// TIA Portal project "JAN0837_proof_of_concept" (V20)

(* hardware
DEVICE "R2D2"  S7-1200 Station
   slot 0: "Rack_0"  S7-1200 Rack  Rack  V1.0
   slot 1: "R2D2_Sharp7"  CPU 1212C DC/DC/DC  6ES7 212-1AE40-0XB0  V4.6
DEVICE "R2D2_1"  S7-1200 Station
   slot 0: "Rack_0"  S7-1200 Rack  Rack  V1.0
   slot 1: "R2D2_OPCUA"  CPU 1212C DC/DC/DC  6ES7 212-1AE40-0XB0  V4.6
DEVICE "R2D2_2"  S7-1200 Station
   slot 0: "Rack_0"  S7-1200 Rack  Rack  V1.0
   slot 1: "R2D2_MQTT"  CPU 1212C DC/DC/DC  6ES7 212-1AE40-0XB0  V4.6
DEVICE "R2D2_3"  S7-1200 Station
   slot 0: "Rack_0"  S7-1200 Rack  Rack  V1.0
   slot 1: "R2D2_MODBUS"  CPU 1212C DC/DC/DC  6ES7 212-1AE40-0XB0  V4.6
DEVICE "R2D2_4"  S7-1200 Station
   slot 0: "Rack_0"  S7-1200 Rack  Rack  V1.0
   slot 1: "R2D2_RESTAPI"  CPU 1212C DC/DC/DC  6ES7 212-1AE40-0XB0  V4.6
*)

// ===== PLC "R2D2_Sharp7"  CPU 1212C DC/DC/DC =====

VAR_GLOBAL   // PLC tag table "Default tag table"
   "Clock_Byte" AT %MB0 : Byte;
   "Clock_10Hz" AT %M0.0 : Bool;
   "Clock_5Hz" AT %M0.1 : Bool;
   "Clock_2.5Hz" AT %M0.2 : Bool;
   "Clock_2Hz" AT %M0.3 : Bool;
   "Clock_1.25Hz" AT %M0.4 : Bool;
   "Clock_1Hz" AT %M0.5 : Bool;
   "Clock_0.625Hz" AT %M0.6 : Bool;
   "Clock_0.5Hz" AT %M0.7 : Bool;
   "System_Byte" AT %MB1 : Byte;
   "FirstScan" AT %M1.0 : Bool;
   "DiagStatusUpdate" AT %M1.1 : Bool;
   "AlwaysTRUE" AT %M1.2 : Bool;
   "AlwaysFALSE" AT %M1.3 : Bool;
END_VAR

VAR_GLOBAL   // PLC tag table "Regulator"
   "Regulator_PV" AT %MD100 : Real;
   "Regulator_SetPoint" AT %MD104 : Real;
END_VAR

VAR_GLOBAL   // PLC tag table "CarLight"
   "CarLight_Tag1" AT %M50.0 : Bool;
END_VAR

VAR_GLOBAL   // PLC tag table "Crossroad"
   "Crossroad_Tag_1" AT %M300.0 : Bool;
   "Crossroad_Tag_2" AT %M300.1 : Bool;
   "Crossroad_Tag_3" AT %MW302 : Word;
   "Crossroad_MEM 0" AT %M304.0 : Bool;
   "Crossroad_MEM 1" AT %M304.1 : Bool;
   "Crossroad_MEM 2" AT %M304.2 : Bool;
   "Crossroad_MEM 3" AT %M304.3 : Bool;
   "Crossroad_MEM 4" AT %M304.4 : Bool;
   "Crossroad_MEM 5" AT %M304.5 : Bool;
   "Crossroad_Clock" AT %MW328 : Int;
   "Crossroad_DayModeState" AT %MB305 : USInt;
   "Crossroad_ActualLengthState" AT %MD316 : Time;
   "Crossorad_HoursDayStart" AT %MW320 : Int;
   "Crossroad_HoursDayEnd" AT %MW322 : Int;
   "Crossroad_DayStarts" AT %MW324 : Int;
   "Crossroad_DayEnds" AT %MW326 : Int;
   "Crossroad_S1" AT %MB306 : USInt;
   "Crossroad_S2" AT %MB307 : USInt;
   "Crossroad_S3" AT %MB308 : USInt;
   "Crossroad_S4" AT %MB309 : USInt;
   "Crossroad_S5" AT %MB310 : USInt;
   "Crossroad_S6" AT %MB311 : USInt;
   "Crossroad_S7" AT %MB312 : USInt;
   "Crossroad_S8" AT %MB313 : USInt;
   "Crossroad_S9" AT %MB314 : USInt;
   "Crossroad_Walk_EN" AT %M330.0 : Bool;
END_VAR

VAR_GLOBAL   // PLC tag table "Crosswalk"
   "Crosswalk_CTU_current_value" AT %MW200 : Int;
   "Crosswalk_CTU_reset" AT %M202.0 : Bool;
   "Crosswalk_DayMode" AT %M202.1 : Bool;
   "Crosswalk_NightMode" AT %M202.2 : Bool;
   "Crosswalk_OffMode" AT %M202.3 : Bool;
   "Crosswalk_DaySeq" AT %MW204 : Int;
   "Crosswalk_NightSeq" AT %MW206 : Int;
END_VAR

TYPE "Crossroad_Input"
   STRUCT
      btnStart : Bool := FALSE;
      btnPause : Bool := FALSE;
      btnStop : Bool := FALSE;
      btnWestCrosswalk1 : Bool := FALSE;
      btnWestCrosswalk2 : Bool := FALSE;
      btnSouthCrosswalk1 : Bool := FALSE;
      btnSouthCrosswalk2 : Bool := FALSE;
      spare1 : DWord := 0;
      spare2 : DWord := 0;
      spare3 : DWord := 0;
      spare4 : DWord := 0;
   END_STRUCT;
END_TYPE

TYPE "Crossroad_Output"
   STRUCT
      crossroadType : Bool := FALSE;
      trafficLightNorth_green : Bool := FALSE;
      trafficLightNorth_yellow : Bool := FALSE;
      trafficLightNorth_red : Bool := FALSE;
      trafficLightSouth_green : Bool := FALSE;
      trafficLightSouth_yellow : Bool := FALSE;
      trafficLightSouth_red : Bool := FALSE;
      trafficLightWest_green : Bool := FALSE;
      trafficLightWest_yellow : Bool := FALSE;
      trafficLightWest_red : Bool := FALSE;
      trafficLightEast_green : Bool := FALSE;
      trafficLightEast_yellow : Bool := FALSE;
      trafficLightEast_red : Bool := FALSE;
      pedestrianSouth1_green : Bool := FALSE;
      pedestrianSouth1_red : Bool := FALSE;
      pedestrianSouth2_green : Bool := FALSE;
      pedestrianSouth2_red : Bool := FALSE;
      pedestrianWest1_green : Bool := FALSE;
      pedestrianWest1_red : Bool := FALSE;
      pedestrianWest2_green : Bool := FALSE;
      pedestrianWest2_red : Bool := FALSE;
      spare1 : DWord := 0;
      spare2 : DWord := 0;
      spare3 : DWord := 0;
      spare4 : DWord := 0;
   END_STRUCT;
END_TYPE

TYPE "Crosswalk_Input"
   STRUCT
      btnStart : Bool := FALSE;
      btnPause : Bool := FALSE;
      btnStop : Bool := FALSE;
      btnCrosswalk1 : Bool := FALSE;
      btnCrosswalk2 : Bool := FALSE;
      spare1 : DWord := 0;
      spare2 : DWord := 0;
      spare3 : DWord := 0;
      spare4 : DWord := 0;
   END_STRUCT;
END_TYPE

TYPE "Crosswalk_Output"
   STRUCT
      crosswalkType : Bool := FALSE;
      trafficLightGreen1 : Bool := FALSE;
      trafficLightsYellow1 : Bool := FALSE;
      trafficLightsRed1 : Bool := FALSE;
      trafficLightGreen2 : Bool := FALSE;
      trafficLightsYellow2 : Bool := FALSE;
      trafficLightsRed2 : Bool := FALSE;
      pedestrianLightGreen1 : Bool := FALSE;
      pedestrianLightRed1 : Bool := FALSE;
      pedestrianLightGreen2 : Bool := FALSE;
      pedestrianLightRed2 : Bool := FALSE;
      spare1 : DWord := 0;
      spare2 : DWord := 0;
      spare3 : DWord := 0;
      spare4 : DWord := 0;
   END_STRUCT;
END_TYPE

TYPE "Regulator_Input"
   STRUCT
      btnReset : Bool := FALSE;
      switchstate : Bool := FALSE;
      order : Int := 1;
      R1 : Real := 0.0;
      R2 : Real := 0.0;
      C1 : Real := 0.0;
      C2 : Real := 0.0;
      Uc1 : Real := 0.0;
      Uc2 : Real := 0.0;
      Td : Real := 0.0;
      Ts : Real := 0.0;
      spare1 : DWord := 0;
      spare2 : DWord := 0;
      spare3 : DWord := 0;
      spare4 : DWord := 0;
   END_STRUCT;
END_TYPE

TYPE "Regulator_Output"
   STRUCT
      Uin : Real := 0.0;
      spare1 : DWord := 0;
      spare2 : DWord := 0;
      spare3 : DWord := 0;
      spare4 : DWord := 0;
   END_STRUCT;
END_TYPE

TYPE "CarLight_Input"
   STRUCT
      btnReset : Bool := FALSE;
      error : Bool := FALSE;
      sensorLight : Bool := FALSE;
      sensorConnectorConnected : Bool := FALSE;
      result : Bool := FALSE;
      spare1 : DWord := 0;
      spare2 : DWord := 0;
      spare3 : DWord := 0;
      spare4 : DWord := 0;
   END_STRUCT;
END_TYPE

TYPE "CarLight_Output"
   STRUCT
      lowBeamLight : Bool := FALSE;
      highBeamLight : Bool := FALSE;
      turnLight : Bool := FALSE;
      spare1 : DWord := 0;
      spare2 : DWord := 0;
      spare3 : DWord := 0;
      spare4 : DWord := 0;
   END_STRUCT;
END_TYPE

DATA_BLOCK "DB_ProcessData"   // DB1
{ S7_Optimized_Access := 'TRUE' }
VERSION : 0.1
   VAR
      crossroad_input : "Crossroad_Input";
      crossroad_output : "Crossroad_Output";
      crosswalk_input : "Crosswalk_Input";
      crosswalk_output : "Crosswalk_Output";
      regulator_input : "Regulator_Input";
      regulator_output : "Regulator_Output";
      carlight_input : "CarLight_Input";
      carlight_output : "CarLight_Output";
   END_VAR
BEGIN
END_DATA_BLOCK

// folder: CarLight

DATA_BLOCK "CarLight_SCL_DB"   // DB12
{ S7_Optimized_Access := 'TRUE' }
VERSION : 0.1
// stored: InstanceOfName CarLight_SCL
"CarLight_SCL"
BEGIN
END_DATA_BLOCK

// folder: System blocks/Program resources

DATA_BLOCK "IEC_Counter_0_DB"   // DB2
{ S7_Optimized_Access := 'TRUE' }
AUTHOR : Simatic
FAMILY : IEC
NAME : CNTR
VERSION : 1.0
// stored: InstanceOfName IEC_COUNTER
"IEC_COUNTER"
BEGIN
END_DATA_BLOCK

DATA_BLOCK "IEC_Timer_0_DB"   // DB3
{ S7_Optimized_Access := 'TRUE' }
AUTHOR : Simatic
FAMILY : IEC
NAME : IEC_TMR
VERSION : 1.0
// stored: InstanceOfName IEC_TIMER
"IEC_TIMER"
BEGIN
END_DATA_BLOCK

DATA_BLOCK "IEC_Timer_CrosswalkGreen_DB_1"   // DB4
{ S7_Optimized_Access := 'TRUE' }
AUTHOR : Simatic
FAMILY : IEC
NAME : IEC_TMR
VERSION : 1.0
// stored: InstanceOfName IEC_TIMER
"IEC_TIMER"
BEGIN
END_DATA_BLOCK

DATA_BLOCK "IEC_Timer_CrosswalkYellow1_DB_1"   // DB5
{ S7_Optimized_Access := 'TRUE' }
AUTHOR : Simatic
FAMILY : IEC
NAME : IEC_TMR
VERSION : 1.0
// stored: InstanceOfName IEC_TIMER
"IEC_TIMER"
BEGIN
END_DATA_BLOCK

DATA_BLOCK "IEC_Timer_CrosswalkRed_DB_1"   // DB6
{ S7_Optimized_Access := 'TRUE' }
AUTHOR : Simatic
FAMILY : IEC
NAME : IEC_TMR
VERSION : 1.0
// stored: InstanceOfName IEC_TIMER
"IEC_TIMER"
BEGIN
END_DATA_BLOCK

DATA_BLOCK "IEC_Timer_CrosswalkYellow2_DB_1"   // DB7
{ S7_Optimized_Access := 'TRUE' }
AUTHOR : Simatic
FAMILY : IEC
NAME : IEC_TMR
VERSION : 1.0
// stored: InstanceOfName IEC_TIMER
"IEC_TIMER"
BEGIN
END_DATA_BLOCK

DATA_BLOCK "IEC_Timer_CrosswalkOn_DB_1"   // DB8
{ S7_Optimized_Access := 'TRUE' }
AUTHOR : Simatic
FAMILY : IEC
NAME : IEC_TMR
VERSION : 1.0
// stored: InstanceOfName IEC_TIMER
"IEC_TIMER"
BEGIN
END_DATA_BLOCK

DATA_BLOCK "IEC_Timer_CrosswalkOff_DB_1"   // DB9
{ S7_Optimized_Access := 'TRUE' }
AUTHOR : Simatic
FAMILY : IEC
NAME : IEC_TMR
VERSION : 1.0
// stored: InstanceOfName IEC_TIMER
"IEC_TIMER"
BEGIN
END_DATA_BLOCK

DATA_BLOCK "IEC_Timer_CrossroadCycle_DB_1"   // DB10
{ S7_Optimized_Access := 'TRUE' }
AUTHOR : Simatic
FAMILY : IEC
NAME : IEC_TMR
VERSION : 1.0
// stored: InstanceOfName IEC_TIMER
"IEC_TIMER"
BEGIN
END_DATA_BLOCK

// folder: (top level)

ORGANIZATION_BLOCK "Main"   // OB1, LAD, ProgramCycle
TITLE = "Main Program Sweep (Cycle)"
{ S7_Optimized_Access := 'TRUE' }
VERSION : 0.1
   VAR_INPUT
      Initial_Call : Bool;   // Initial call of this OB
      Remanence : Bool;   // =True, if remanent data are available
   END_VAR
BEGIN

REGION Network 1: CarLight
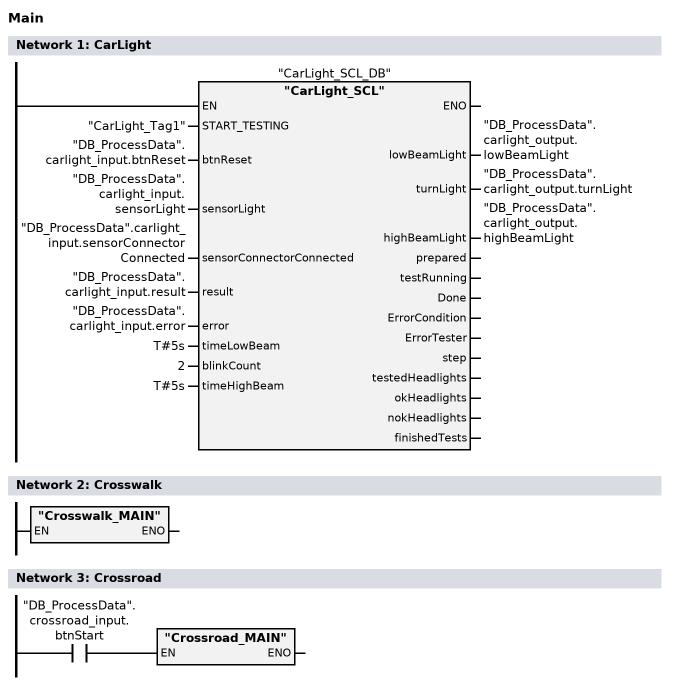
   RUNG wire#powerrail
      "CarLight_SCL_DB"(START_TESTING := "CarLight_Tag1", btnReset := "DB_ProcessData".carlight_input.btnReset, sensorLight := "DB_ProcessData".carlight_input.sensorLight, sensorConnectorConnected := "DB_ProcessData".carlight_input.sensorConnectorConnected, result := "DB_ProcessData".carlight_input.result, error := "DB_ProcessData".carlight_input.error, timeLowBeam := T#5s, blinkCount := 2, timeHighBeam := T#5s, lowBeamLight => "DB_ProcessData".carlight_output.lowBeamLight, turnLight => "DB_ProcessData".carlight_output.turnLight, highBeamLight => "DB_ProcessData".carlight_output.highBeamLight, prepared =>, testRunning =>, Done =>, ErrorCondition =>, ErrorTester =>, "step" =>, testedHeadlights =>, okHeadlights =>, nokHeadlights =>, finishedTests =>)
   END_RUNG
   // the same network as SCL:
   "CarLight_SCL_DB"(START_TESTING := "CarLight_Tag1",   // "CarLight_SCL"
                     btnReset := "DB_ProcessData".carlight_input.btnReset,
                     sensorLight := "DB_ProcessData".carlight_input.sensorLight,
                     sensorConnectorConnected := "DB_ProcessData".carlight_input.sensorConnectorConnected,
                     result := "DB_ProcessData".carlight_input.result,
                     error := "DB_ProcessData".carlight_input.error,
                     timeLowBeam := T#5s,
                     blinkCount := 2,
                     timeHighBeam := T#5s,
                     lowBeamLight => "DB_ProcessData".carlight_output.lowBeamLight,
                     turnLight => "DB_ProcessData".carlight_output.turnLight,
                     highBeamLight => "DB_ProcessData".carlight_output.highBeamLight);
END_REGION

REGION Network 2: Crosswalk
   RUNG wire#powerrail
      "Crosswalk_MAIN"()
   END_RUNG
   // the same network as SCL:
   "Crosswalk_MAIN"();
END_REGION

REGION Network 3: Crossroad
   RUNG wire#powerrail
      Contact( "DB_ProcessData".crossroad_input.btnStart )
      "Crossroad_MAIN"()
   END_RUNG
   // the same network as SCL:
   IF "DB_ProcessData".crossroad_input.btnStart THEN "Crossroad_MAIN"(); END_IF;
END_REGION
END_ORGANIZATION_BLOCK

ORGANIZATION_BLOCK "CyclicInterrupt"   // OB30, LAD, CyclicInterrupt
{ S7_Optimized_Access := 'TRUE' }
VERSION : 0.1
   VAR_INPUT
      Initial_Call : Bool;   // Initial call of this OB
      Event_Count : Int;   // Events discarded
   END_VAR
BEGIN

REGION Network 1: Regulator
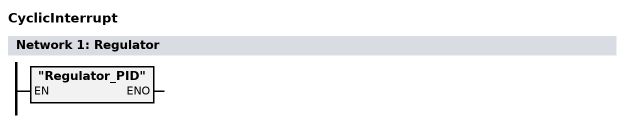
   RUNG wire#powerrail
      "Regulator_PID"()
   END_RUNG
   // the same network as SCL:
   "Regulator_PID"();
END_REGION
END_ORGANIZATION_BLOCK

ORGANIZATION_BLOCK "Startup"   // OB100, LAD, Startup
TITLE = "Complete Restart"
{ S7_Optimized_Access := 'TRUE' }
VERSION : 0.1
   VAR_INPUT
      LostRetentive : Bool;   // True if retentive data are lost
      LostRTC : Bool;   // True if date and time are lost
   END_VAR
BEGIN

REGION Network 1 (SCL)
   // Communication 


   // Crossroad
   "Crossorad_HoursDayStart" := 0;
   "Crossroad_HoursDayEnd" := 2400;
   "Crossroad_DayStarts" := 500;
   "Crossroad_DayEnds" := 2200;
   "Crossroad_S1" := 1;
   "Crossroad_S2" := 2;
   "Crossroad_S3" := 3;
   "Crossroad_S4" := 4;
   "Crossroad_S5" := 5;
   "Crossroad_S6" := 6;
   "Crossroad_S7" := 7;
   "Crossroad_S8" := 8;
   "Crossroad_S9" := 9;


   // Crosswalk


   // Regulaotr


   // CarLight
END_REGION
END_ORGANIZATION_BLOCK

// folder: CarLight

FUNCTION_BLOCK "CarLight_SCL"   // FB1, SCL
{ S7_Optimized_Access := 'TRUE' }
VERSION : 0.1
   VAR_INPUT
      START_TESTING : Bool;
      btnReset : Bool;
      sensorLight : Bool;
      sensorConnectorConnected : Bool;
      result : Bool;
      error : Bool;
      timeLowBeam : Time;
      blinkCount : Int;
      timeHighBeam : Time;
   END_VAR
   VAR_OUTPUT
      lowBeamLight : Bool;
      turnLight : Bool;
      highBeamLight : Bool;
      prepared : Bool;
      testRunning : Bool;
      Done : Bool;
      ErrorCondition : Bool;
      ErrorTester : Bool;
      "step" : Int;
      testedHeadlights : DInt;
      okHeadlights : DInt;
      nokHeadlights : DInt;
      finishedTests : DInt;
   END_VAR
   VAR
      state : Int;
      ready : Bool;
      start_old : Bool;
      start_rise : Bool;
      conditionsErrorLatched : Bool;
      testerErrorLatched : Bool;
      blinkTarget : Int;
      blinkIndex : Int;
      resultStored : Bool;
      testerResponseSeenTrue : Bool;
      tonLowBeam : TON_TIME;
      tonBlinkOn : TON_TIME;
      tonBlinkOff : TON_TIME;
      tonHighBeam : TON_TIME;
      tonAll : TON_TIME;
      tonTesterResponse : TON_TIME;
   END_VAR
BEGIN
   // ---------------------------------------------------------------------
   // Helper signals
   // ---------------------------------------------------------------------
   #ready := #sensorLight AND #sensorConnectorConnected;

   IF #blinkCount < 1 THEN
       #blinkTarget := 1;
   ELSE
       #blinkTarget := #blinkCount;
   END_IF;

   #start_rise := #START_TESTING AND NOT #start_old;
   #start_old := #START_TESTING;


   // ---------------------------------------------------------------------
   // RESET process (counters are NOT cleared)
   // ---------------------------------------------------------------------
   IF #btnReset THEN
       #state := 0;
       #conditionsErrorLatched := FALSE;
       #testerErrorLatched := FALSE;   
       #blinkIndex := 0;
       #resultStored := FALSE;
       #testerResponseSeenTrue := FALSE;
   END_IF;


   // ---------------------------------------------------------------------
   // Loss of required conditions during test
   // ---------------------------------------------------------------------
   IF ((#state >= 20) AND (#state <= 55)) AND (NOT #ready) THEN
       #state := 0;
       #conditionsErrorLatched := TRUE;
       #blinkIndex := 0;
       #resultStored := FALSE;
       #testerResponseSeenTrue := FALSE;
   END_IF;


   // ---------------------------------------------------------------------
   // Tester error – immediate NOK termination
   // ---------------------------------------------------------------------
   IF ((#state >= 20) AND (#state <= 55)) AND #error THEN

       #testerErrorLatched := TRUE;

       IF NOT #resultStored THEN
           #testedHeadlights := #testedHeadlights + 1;
           #nokHeadlights := #nokHeadlights + 1;
           #resultStored := TRUE;
       END_IF;

       #blinkIndex := 0;
       #testerResponseSeenTrue := FALSE;

       #state := 70;

   END_IF;


   // ---------------------------------------------------------------------
   // State machine
   // ---------------------------------------------------------------------
   CASE #state OF


           // ==============================================================
           // 0 - IDLE
           // ==============================================================
       0:

           #lowBeamLight := FALSE;
           #turnLight := FALSE;
           #highBeamLight := FALSE;

           #tonLowBeam(IN := FALSE,
                     PT := #timeLowBeam);
           #tonBlinkOn(IN := FALSE,
                       PT := T#1s);
           #tonBlinkOff(IN := FALSE,
                        PT := T#1s);
           #tonHighBeam(IN := FALSE,
                     PT := #timeHighBeam);
           #tonAll(IN := FALSE,
                   PT := T#5s);
           #tonTesterResponse(IN := FALSE,
                              PT := T#1s);

           IF #start_rise THEN

               IF #ready AND (NOT #error) THEN

                   #conditionsErrorLatched := FALSE;
                   #testerErrorLatched := FALSE;
                   #blinkIndex := 0;
                   #resultStored := FALSE;
                   #testerResponseSeenTrue := FALSE;

                   #state := 20;

               ELSE

                   IF NOT #ready THEN
                       #conditionsErrorLatched := TRUE;
                   END_IF;

                   IF #error THEN
                       #testerErrorLatched := TRUE;
                   END_IF;

               END_IF;

           END_IF;


           // ==============================================================
           // 20 - LOW BEAM
           // ==============================================================
       20:

           #lowBeamLight := TRUE;
           #turnLight := FALSE;
           #highBeamLight := FALSE;

           #tonLowBeam(IN := TRUE,
                     PT := #timeLowBeam);
           #tonBlinkOn(IN := FALSE,
                       PT := T#1s);
           #tonBlinkOff(IN := FALSE,
                        PT := T#1s);
           #tonHighBeam(IN := FALSE,
                     PT := #timeHighBeam);
           #tonAll(IN := FALSE,
                   PT := T#5s);
           #tonTesterResponse(IN := FALSE,
                              PT := T#1s);

           IF #tonLowBeam.Q THEN
               #blinkIndex := 0;
               #state := 30;
           END_IF;


           // ==============================================================
           // 30 - TURN SIGNAL ON
           // ==============================================================
       30:

           #lowBeamLight := FALSE;
           #turnLight := TRUE;
           #highBeamLight := FALSE;

           #tonLowBeam(IN := FALSE,
                     PT := #timeLowBeam);
           #tonBlinkOn(IN := TRUE,
                       PT := T#1s);
           #tonBlinkOff(IN := FALSE,
                        PT := T#1s);
           #tonHighBeam(IN := FALSE,
                     PT := #timeHighBeam);
           #tonAll(IN := FALSE,
                   PT := T#5s);
           #tonTesterResponse(IN := FALSE,
                              PT := T#1s);

           IF #tonBlinkOn.Q THEN
               #state := 31;
           END_IF;


           // ==============================================================
           // 31 - TURN SIGNAL OFF
           // ==============================================================
       31:

           #lowBeamLight := FALSE;
           #turnLight := FALSE;
           #highBeamLight := FALSE;

           #tonLowBeam(IN := FALSE,
                     PT := #timeLowBeam);
           #tonBlinkOn(IN := FALSE,
                       PT := T#1s);
           #tonBlinkOff(IN := TRUE,
                        PT := T#1s);
           #tonHighBeam(IN := FALSE,
                     PT := #timeHighBeam);
           #tonAll(IN := FALSE,
                   PT := T#5s);
           #tonTesterResponse(IN := FALSE,
                              PT := T#1s);

           IF #tonBlinkOff.Q THEN

               #blinkIndex := #blinkIndex + 1;

               IF #blinkIndex < #blinkTarget THEN
                   #state := 30;
               ELSE
                   #state := 40;
               END_IF;

           END_IF;


           // ==============================================================
           // 40 - HIGH BEAM
           // ==============================================================
       40:

           #lowBeamLight := FALSE;
           #turnLight := FALSE;
           #highBeamLight := TRUE;

           #tonLowBeam(IN := FALSE,
                     PT := #timeLowBeam);
           #tonBlinkOn(IN := FALSE,
                       PT := T#1s);
           #tonBlinkOff(IN := FALSE,
                        PT := T#1s);
           #tonHighBeam(IN := TRUE,
                     PT := #timeHighBeam);
           #tonAll(IN := FALSE,
                   PT := T#5s);
           #tonTesterResponse(IN := FALSE,
                              PT := T#1s);

           IF #tonHighBeam.Q THEN
               #state := 50;
           END_IF;


           // ==============================================================
           // 50 - ALL LIGHTS (5 seconds)
           // ==============================================================
       50:

           #lowBeamLight := TRUE;
           #turnLight := TRUE;
           #highBeamLight := TRUE;

           #tonLowBeam(IN := FALSE,
                     PT := #timeLowBeam);
           #tonBlinkOn(IN := FALSE,
                       PT := T#1s);
           #tonBlinkOff(IN := FALSE,
                        PT := T#1s);
           #tonHighBeam(IN := FALSE,
                     PT := #timeHighBeam);
           #tonAll(IN := TRUE,
                   PT := T#5s);
           #tonTesterResponse(IN := FALSE,
                              PT := T#1s);

           IF #tonAll.Q THEN
               #testerResponseSeenTrue := FALSE;
               #state := 55;
           END_IF;


           // ==============================================================
           // 55 - WAIT 1 s FOR RESULT
           // ==============================================================
       55:

           #lowBeamLight := FALSE;
           #turnLight := FALSE;
           #highBeamLight := FALSE;

           #tonLowBeam(IN := FALSE,
                     PT := #timeLowBeam);
           #tonBlinkOn(IN := FALSE,
                       PT := T#1s);
           #tonBlinkOff(IN := FALSE,
                        PT := T#1s);
           #tonHighBeam(IN := FALSE,
                     PT := #timeHighBeam);
           #tonAll(IN := FALSE,
                   PT := T#5s);
           #tonTesterResponse(IN := TRUE,
                              PT := T#1s);

           IF #result THEN
               #testerResponseSeenTrue := TRUE;
           END_IF;

           IF #tonTesterResponse.Q THEN

               IF NOT #resultStored THEN

                   #testedHeadlights := #testedHeadlights + 1;

                   IF #testerResponseSeenTrue THEN
                       #okHeadlights := #okHeadlights + 1;
                   ELSE
                       #nokHeadlights := #nokHeadlights + 1;
                   END_IF;

                   #resultStored := TRUE;

               END_IF;

               #finishedTests := #finishedTests + 1;

               #state := 60;

           END_IF;


           // ==============================================================
           // 60 - FINISHED
           // ==============================================================
       60:

           #lowBeamLight := FALSE;
           #turnLight := FALSE;
           #highBeamLight := FALSE;

           IF #start_rise THEN

               IF #ready AND (NOT #error) THEN

                   #conditionsErrorLatched := FALSE;
                   #testerErrorLatched := FALSE;
                   #blinkIndex := 0;
                   #resultStored := FALSE;
                   #testerResponseSeenTrue := FALSE;

                   #state := 20;

               END_IF;

           END_IF;


           // ==============================================================
           // 70 - TESTER ERROR
           // ==============================================================
       70:

           #lowBeamLight := FALSE;
           #turnLight := FALSE;
           #highBeamLight := FALSE;

           IF #start_rise THEN

               IF #ready AND (NOT #error) THEN

                   #conditionsErrorLatched := FALSE;
                   #testerErrorLatched := FALSE;
                   #blinkIndex := 0;
                   #resultStored := FALSE;
                   #testerResponseSeenTrue := FALSE;

                   #state := 20;

               END_IF;

           END_IF;

       ELSE

           #state := 0;

   END_CASE;


   // ---------------------------------------------------------------------
   // State outputs
   // ---------------------------------------------------------------------
   #testRunning := (#state >= 20) AND (#state <= 55);

   #prepared := #ready AND (NOT #error) AND
   ((#state = 0) OR (#state = 60) OR (#state = 70));

   #Done := (#state = 60);

   #ErrorCondition := #conditionsErrorLatched;
   #ErrorTester := #testerErrorLatched;

   #step := #state;
END_FUNCTION_BLOCK

// folder: Crossroad

FUNCTION "Crossroad_MAIN" : Void   // FC4, LAD
{ S7_Optimized_Access := 'TRUE' }
VERSION : 0.1
   VAR_TEMP   // added for the SCL form of the ladder/FBD networks
      _w1 : Bool;
      _w2 : Bool;
      _w3 : Bool;
      _w4 : Bool;
   END_VAR
BEGIN

REGION Network 1: Time based decision process
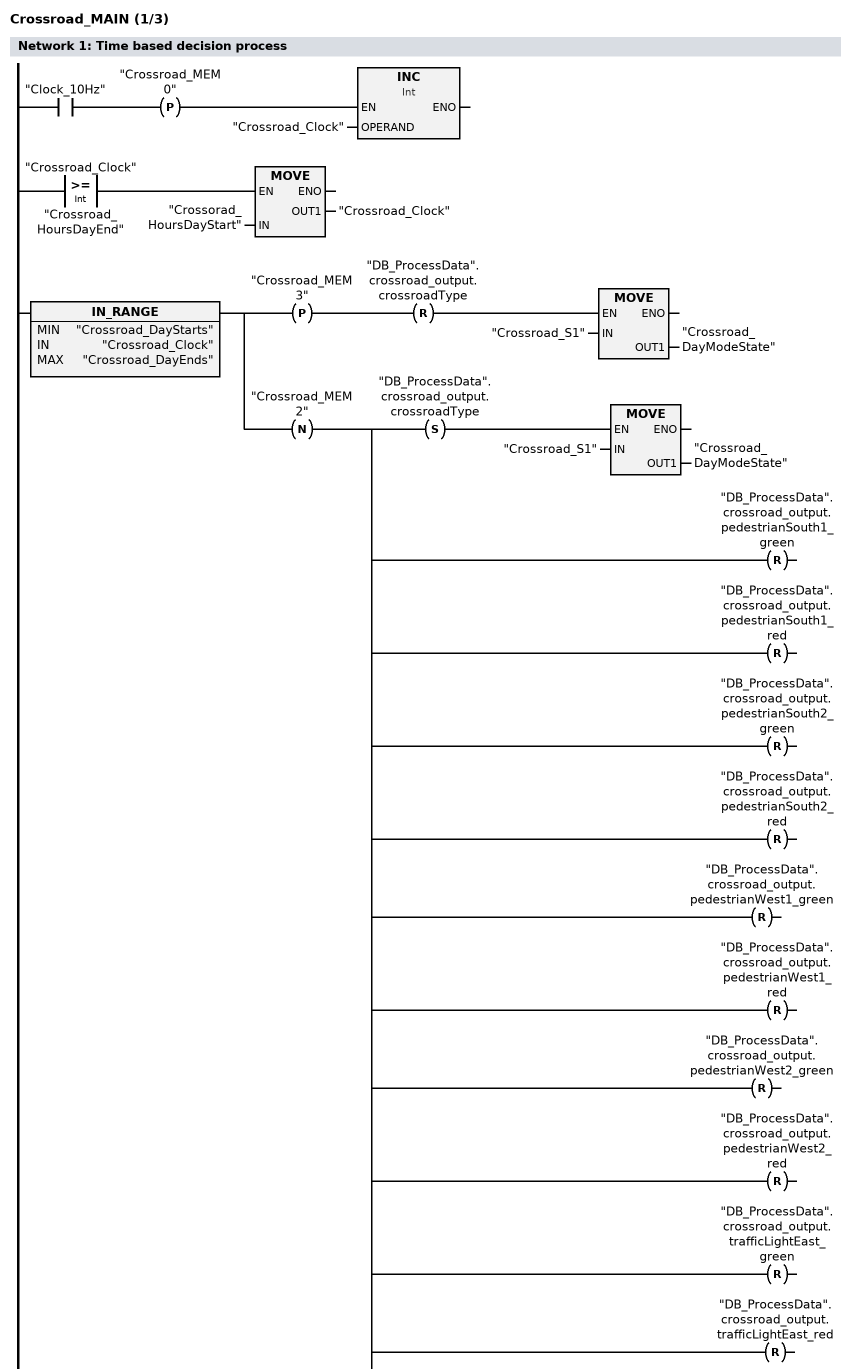
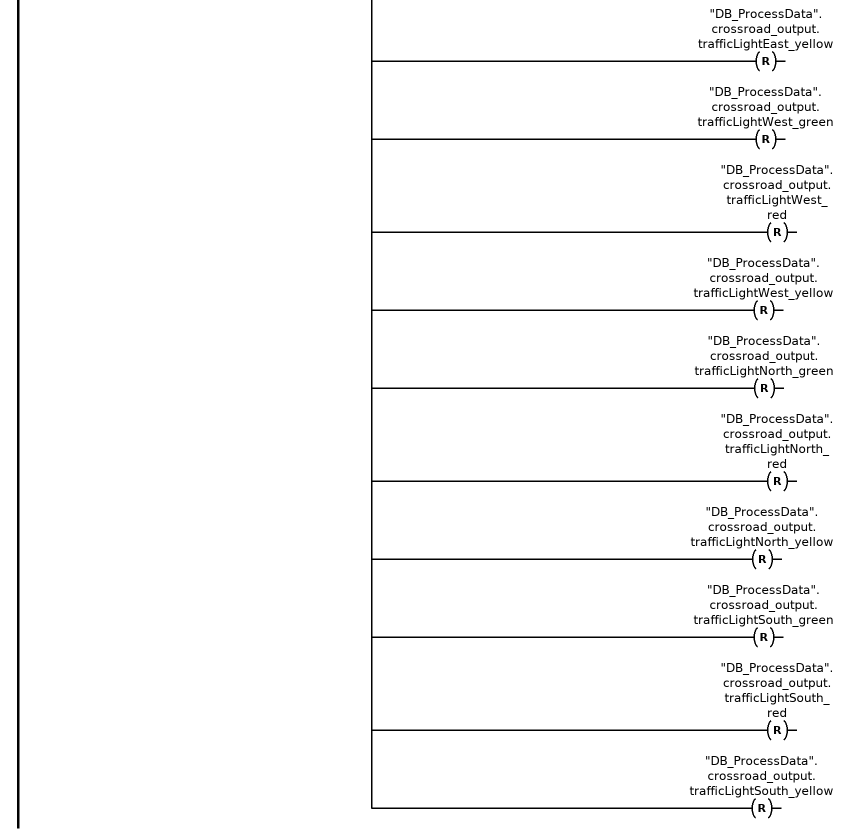
   RUNG wire#powerrail
      Contact( "Clock_10Hz" )
      P_Trig( "Crossroad_MEM 0" )
      { S7_Templates := "DestType := Int" } Inc( "Crossroad_Clock" )
   END_RUNG
   RUNG wire#powerrail
      { S7_Templates := "SrcType := Int" } GE_Contact(in1 := "Crossroad_Clock", in2 := "Crossroad_HoursDayEnd")
      Move(in := "Crossorad_HoursDayStart", out1 => "Crossroad_Clock")
   END_RUNG
   RUNG wire#powerrail
      { S7_Templates := "SrcType := Int" } InRange(min := "Crossroad_DayStarts", in := "Crossroad_Clock", max := "Crossroad_DayEnds")
      wire#w1
      P_Trig( "Crossroad_MEM 3" )
      R_Coil( "DB_ProcessData".crossroad_output.crossroadType )
      Move(in := "Crossroad_S1", out1 => "Crossroad_DayModeState")
   END_RUNG
   RUNG wire#w1
      N_Trig( "Crossroad_MEM 2" )
      wire#w2
      S_Coil( "DB_ProcessData".crossroad_output.crossroadType )
      Move(in := "Crossroad_S1", out1 => "Crossroad_DayModeState")
   END_RUNG
   RUNG wire#w2
      R_Coil( "DB_ProcessData".crossroad_output.pedestrianSouth1_green )
   END_RUNG
   RUNG wire#w2
      R_Coil( "DB_ProcessData".crossroad_output.pedestrianSouth1_red )
   END_RUNG
   RUNG wire#w2
      R_Coil( "DB_ProcessData".crossroad_output.pedestrianSouth2_green )
   END_RUNG
   RUNG wire#w2
      R_Coil( "DB_ProcessData".crossroad_output.pedestrianSouth2_red )
   END_RUNG
   RUNG wire#w2
      R_Coil( "DB_ProcessData".crossroad_output.pedestrianWest1_green )
   END_RUNG
   RUNG wire#w2
      R_Coil( "DB_ProcessData".crossroad_output.pedestrianWest1_red )
   END_RUNG
   RUNG wire#w2
      R_Coil( "DB_ProcessData".crossroad_output.pedestrianWest2_green )
   END_RUNG
   RUNG wire#w2
      R_Coil( "DB_ProcessData".crossroad_output.pedestrianWest2_red )
   END_RUNG
   RUNG wire#w2
      R_Coil( "DB_ProcessData".crossroad_output.trafficLightEast_green )
   END_RUNG
   RUNG wire#w2
      R_Coil( "DB_ProcessData".crossroad_output.trafficLightEast_red )
   END_RUNG
   RUNG wire#w2
      R_Coil( "DB_ProcessData".crossroad_output.trafficLightEast_yellow )
   END_RUNG
   RUNG wire#w2
      R_Coil( "DB_ProcessData".crossroad_output.trafficLightWest_green )
   END_RUNG
   RUNG wire#w2
      R_Coil( "DB_ProcessData".crossroad_output.trafficLightWest_red )
   END_RUNG
   RUNG wire#w2
      R_Coil( "DB_ProcessData".crossroad_output.trafficLightWest_yellow )
   END_RUNG
   RUNG wire#w2
      R_Coil( "DB_ProcessData".crossroad_output.trafficLightNorth_green )
   END_RUNG
   RUNG wire#w2
      R_Coil( "DB_ProcessData".crossroad_output.trafficLightNorth_red )
   END_RUNG
   RUNG wire#w2
      R_Coil( "DB_ProcessData".crossroad_output.trafficLightNorth_yellow )
   END_RUNG
   RUNG wire#w2
      R_Coil( "DB_ProcessData".crossroad_output.trafficLightSouth_green )
   END_RUNG
   RUNG wire#w2
      R_Coil( "DB_ProcessData".crossroad_output.trafficLightSouth_red )
   END_RUNG
   RUNG wire#w2
      R_Coil( "DB_ProcessData".crossroad_output.trafficLightSouth_yellow )
   END_RUNG
   // the same network as SCL:
   #_w1 := "Clock_10Hz" AND NOT "Crossroad_MEM 0";   // rising edge
   "Crossroad_MEM 0" := "Clock_10Hz";
   IF #_w1 THEN "Crossroad_Clock" := "Crossroad_Clock" + 1; END_IF;
   IF "Crossroad_Clock" >= "Crossroad_HoursDayEnd" THEN
       "Crossroad_Clock" := "Crossorad_HoursDayStart";
   END_IF;
   #_w2 := ("Crossroad_DayStarts" <= "Crossroad_Clock") AND ("Crossroad_Clock" <= "Crossroad_DayEnds");
   #_w3 := #_w2 AND NOT "Crossroad_MEM 3";   // rising edge
   "Crossroad_MEM 3" := #_w2;
   IF #_w3 THEN
       "DB_ProcessData".crossroad_output.crossroadType := FALSE;
       "Crossroad_DayModeState" := "Crossroad_S1";
   END_IF;
   #_w4 := NOT #_w2 AND "Crossroad_MEM 2";   // falling edge
   "Crossroad_MEM 2" := #_w2;
   IF #_w4 THEN
       "DB_ProcessData".crossroad_output.crossroadType := TRUE;
       "Crossroad_DayModeState" := "Crossroad_S1";
       "DB_ProcessData".crossroad_output.pedestrianSouth1_green := FALSE;
       "DB_ProcessData".crossroad_output.pedestrianSouth1_red := FALSE;
       "DB_ProcessData".crossroad_output.pedestrianSouth2_green := FALSE;
       "DB_ProcessData".crossroad_output.pedestrianSouth2_red := FALSE;
       "DB_ProcessData".crossroad_output.pedestrianWest1_green := FALSE;
       "DB_ProcessData".crossroad_output.pedestrianWest1_red := FALSE;
       "DB_ProcessData".crossroad_output.pedestrianWest2_green := FALSE;
       "DB_ProcessData".crossroad_output.pedestrianWest2_red := FALSE;
       "DB_ProcessData".crossroad_output.trafficLightEast_green := FALSE;
       "DB_ProcessData".crossroad_output.trafficLightEast_red := FALSE;
       "DB_ProcessData".crossroad_output.trafficLightEast_yellow := FALSE;
       "DB_ProcessData".crossroad_output.trafficLightWest_green := FALSE;
       "DB_ProcessData".crossroad_output.trafficLightWest_red := FALSE;
       "DB_ProcessData".crossroad_output.trafficLightWest_yellow := FALSE;
       "DB_ProcessData".crossroad_output.trafficLightNorth_green := FALSE;
       "DB_ProcessData".crossroad_output.trafficLightNorth_red := FALSE;
       "DB_ProcessData".crossroad_output.trafficLightNorth_yellow := FALSE;
       "DB_ProcessData".crossroad_output.trafficLightSouth_green := FALSE;
       "DB_ProcessData".crossroad_output.trafficLightSouth_red := FALSE;
       "DB_ProcessData".crossroad_output.trafficLightSouth_yellow := FALSE;
   END_IF;
END_REGION

REGION Network 2: Night mode
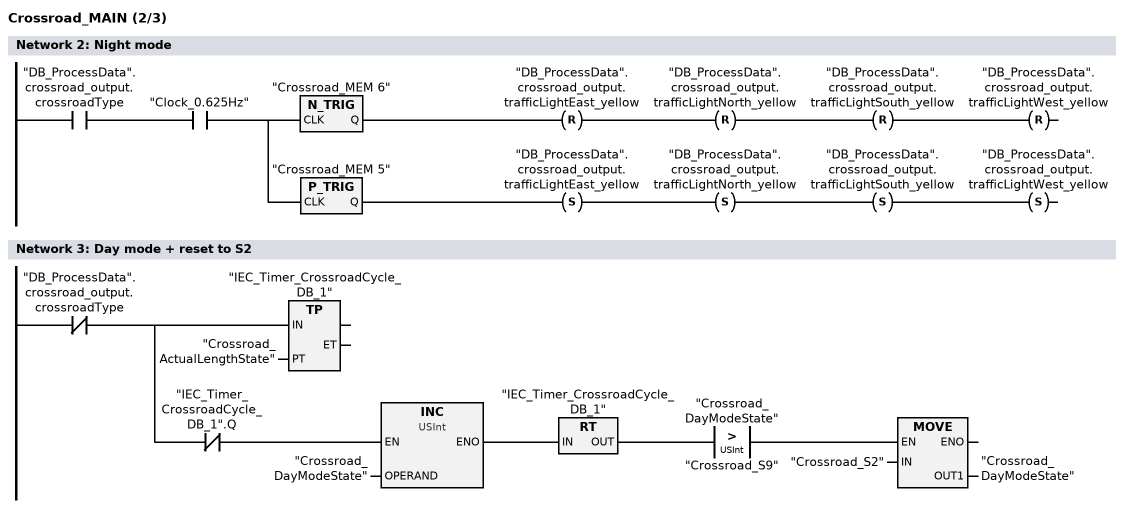
   RUNG wire#powerrail
      Contact( "DB_ProcessData".crossroad_output.crossroadType )
      Contact( "Clock_0.625Hz" )
      wire#w1
      N_Trig( "Crossroad_MEM 6" )
      R_Coil( "DB_ProcessData".crossroad_output.trafficLightEast_yellow )
      R_Coil( "DB_ProcessData".crossroad_output.trafficLightNorth_yellow )
      R_Coil( "DB_ProcessData".crossroad_output.trafficLightSouth_yellow )
      R_Coil( "DB_ProcessData".crossroad_output.trafficLightWest_yellow )
   END_RUNG
   RUNG wire#w1
      P_Trig( "Crossroad_MEM 5" )
      S_Coil( "DB_ProcessData".crossroad_output.trafficLightEast_yellow )
      S_Coil( "DB_ProcessData".crossroad_output.trafficLightNorth_yellow )
      S_Coil( "DB_ProcessData".crossroad_output.trafficLightSouth_yellow )
      S_Coil( "DB_ProcessData".crossroad_output.trafficLightWest_yellow )
   END_RUNG
   // the same network as SCL:
   #_w1 := "DB_ProcessData".crossroad_output.crossroadType AND "Clock_0.625Hz";
   #_w2 := NOT #_w1 AND "Crossroad_MEM 6";   // falling edge
   "Crossroad_MEM 6" := #_w1;
   IF #_w2 THEN
       "DB_ProcessData".crossroad_output.trafficLightEast_yellow := FALSE;
       "DB_ProcessData".crossroad_output.trafficLightNorth_yellow := FALSE;
       "DB_ProcessData".crossroad_output.trafficLightSouth_yellow := FALSE;
       "DB_ProcessData".crossroad_output.trafficLightWest_yellow := FALSE;
   END_IF;
   #_w3 := #_w1 AND NOT "Crossroad_MEM 5";   // rising edge
   "Crossroad_MEM 5" := #_w1;
   IF #_w3 THEN
       "DB_ProcessData".crossroad_output.trafficLightEast_yellow := TRUE;
       "DB_ProcessData".crossroad_output.trafficLightNorth_yellow := TRUE;
       "DB_ProcessData".crossroad_output.trafficLightSouth_yellow := TRUE;
       "DB_ProcessData".crossroad_output.trafficLightWest_yellow := TRUE;
   END_IF;
END_REGION

REGION Network 3: Day mode + reset to S2
   #_w1 := NOT "DB_ProcessData".crossroad_output.crossroadType;
   "IEC_Timer_CrossroadCycle_DB_1".TP(IN := #_w1, PT := "Crossroad_ActualLengthState");
   #_w2 := #_w1 AND NOT "IEC_Timer_CrossroadCycle_DB_1".Q;
   IF #_w2 THEN
       "Crossroad_DayModeState" := "Crossroad_DayModeState" + 1;
       RESET_TIMER("IEC_Timer_CrossroadCycle_DB_1");
   END_IF;
   IF #_w2 AND ("Crossroad_DayModeState" > "Crossroad_S9") THEN
       "Crossroad_DayModeState" := "Crossroad_S2";
   END_IF;
END_REGION

REGION Network 4: Day mode time seq
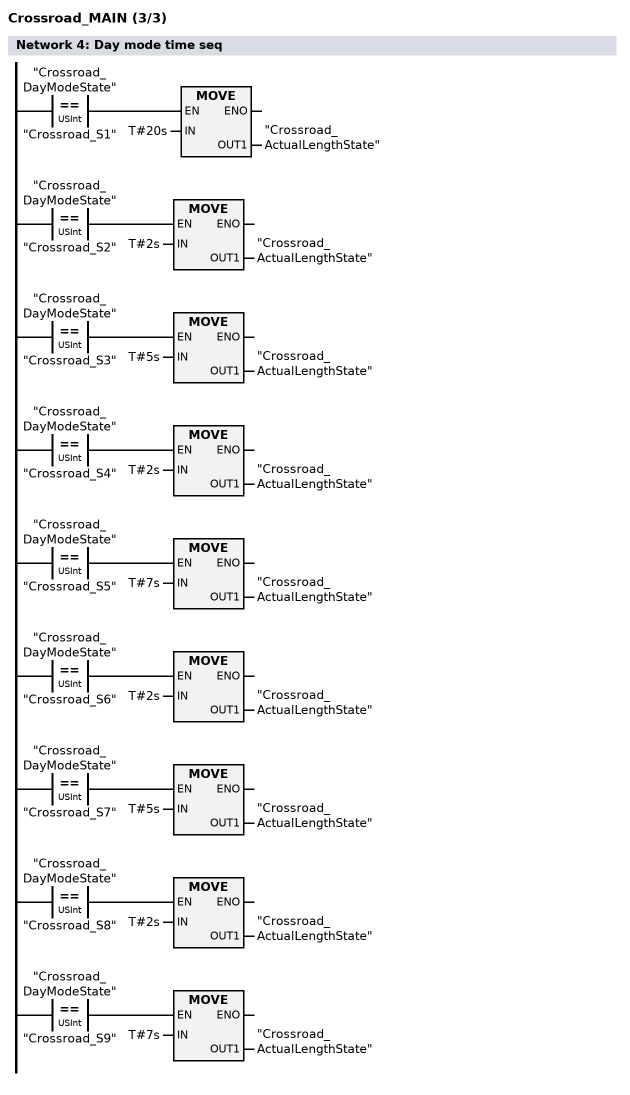
   RUNG wire#powerrail
      { S7_Templates := "SrcType := USInt" } EQ_Contact(in1 := "Crossroad_DayModeState", in2 := "Crossroad_S1")
      Move(in := T#20s, out1 => "Crossroad_ActualLengthState")
   END_RUNG
   RUNG wire#powerrail
      { S7_Templates := "SrcType := USInt" } EQ_Contact(in1 := "Crossroad_DayModeState", in2 := "Crossroad_S2")
      Move(in := T#2s, out1 => "Crossroad_ActualLengthState")
   END_RUNG
   RUNG wire#powerrail
      { S7_Templates := "SrcType := USInt" } EQ_Contact(in1 := "Crossroad_DayModeState", in2 := "Crossroad_S3")
      Move(in := T#5s, out1 => "Crossroad_ActualLengthState")
   END_RUNG
   RUNG wire#powerrail
      { S7_Templates := "SrcType := USInt" } EQ_Contact(in1 := "Crossroad_DayModeState", in2 := "Crossroad_S4")
      Move(in := T#2s, out1 => "Crossroad_ActualLengthState")
   END_RUNG
   RUNG wire#powerrail
      { S7_Templates := "SrcType := USInt" } EQ_Contact(in1 := "Crossroad_DayModeState", in2 := "Crossroad_S5")
      Move(in := T#7s, out1 => "Crossroad_ActualLengthState")
   END_RUNG
   RUNG wire#powerrail
      { S7_Templates := "SrcType := USInt" } EQ_Contact(in1 := "Crossroad_DayModeState", in2 := "Crossroad_S6")
      Move(in := T#2s, out1 => "Crossroad_ActualLengthState")
   END_RUNG
   RUNG wire#powerrail
      { S7_Templates := "SrcType := USInt" } EQ_Contact(in1 := "Crossroad_DayModeState", in2 := "Crossroad_S7")
      Move(in := T#5s, out1 => "Crossroad_ActualLengthState")
   END_RUNG
   RUNG wire#powerrail
      { S7_Templates := "SrcType := USInt" } EQ_Contact(in1 := "Crossroad_DayModeState", in2 := "Crossroad_S8")
      Move(in := T#2s, out1 => "Crossroad_ActualLengthState")
   END_RUNG
   RUNG wire#powerrail
      { S7_Templates := "SrcType := USInt" } EQ_Contact(in1 := "Crossroad_DayModeState", in2 := "Crossroad_S9")
      Move(in := T#7s, out1 => "Crossroad_ActualLengthState")
   END_RUNG
   // the same network as SCL:
   IF "Crossroad_DayModeState" = "Crossroad_S1" THEN "Crossroad_ActualLengthState" := T#20s; END_IF;
   IF "Crossroad_DayModeState" = "Crossroad_S2" THEN "Crossroad_ActualLengthState" := T#2s; END_IF;
   IF "Crossroad_DayModeState" = "Crossroad_S3" THEN "Crossroad_ActualLengthState" := T#5s; END_IF;
   IF "Crossroad_DayModeState" = "Crossroad_S4" THEN "Crossroad_ActualLengthState" := T#2s; END_IF;
   IF "Crossroad_DayModeState" = "Crossroad_S5" THEN "Crossroad_ActualLengthState" := T#7s; END_IF;
   IF "Crossroad_DayModeState" = "Crossroad_S6" THEN "Crossroad_ActualLengthState" := T#2s; END_IF;
   IF "Crossroad_DayModeState" = "Crossroad_S7" THEN "Crossroad_ActualLengthState" := T#5s; END_IF;
   IF "Crossroad_DayModeState" = "Crossroad_S8" THEN "Crossroad_ActualLengthState" := T#2s; END_IF;
   IF "Crossroad_DayModeState" = "Crossroad_S9" THEN "Crossroad_ActualLengthState" := T#7s; END_IF;
END_REGION

REGION Network 5 (SCL): Day mode lights
   IF NOT "DB_ProcessData".crossroad_output.crossroadType THEN
       CASE "Crossroad_DayModeState" OF
           1:  // Statement section case S1
               // GREEN = FALSE, YELLOW = FALSE, RED = TRUE
               // PED: RED = TRUE, GREEN = FALSE

               "DB_ProcessData".crossroad_output.trafficLightEast_green := FALSE;
               "DB_ProcessData".crossroad_output.trafficLightEast_red := TRUE;
               "DB_ProcessData".crossroad_output.trafficLightEast_yellow := FALSE;

               "DB_ProcessData".crossroad_output.trafficLightNorth_green := FALSE;
               "DB_ProcessData".crossroad_output.trafficLightNorth_red := TRUE;
               "DB_ProcessData".crossroad_output.trafficLightNorth_yellow := FALSE;

               "DB_ProcessData".crossroad_output.trafficLightSouth_green := FALSE;
               "DB_ProcessData".crossroad_output.trafficLightSouth_red := TRUE;
               "DB_ProcessData".crossroad_output.trafficLightSouth_yellow := FALSE;

               "DB_ProcessData".crossroad_output.trafficLightWest_green := FALSE;
               "DB_ProcessData".crossroad_output.trafficLightWest_red := TRUE;
               "DB_ProcessData".crossroad_output.trafficLightWest_yellow := FALSE;

               "DB_ProcessData".crossroad_output.pedestrianSouth1_green := FALSE;
               "DB_ProcessData".crossroad_output.pedestrianSouth1_red := TRUE;
               "DB_ProcessData".crossroad_output.pedestrianSouth2_green := FALSE;
               "DB_ProcessData".crossroad_output.pedestrianSouth2_red := TRUE;

               "DB_ProcessData".crossroad_output.pedestrianWest1_green := FALSE;
               "DB_ProcessData".crossroad_output.pedestrianWest1_red := TRUE;
               "DB_ProcessData".crossroad_output.pedestrianWest2_green := FALSE;
               "DB_ProcessData".crossroad_output.pedestrianWest2_red := TRUE;

               //"PLC_LED_GREEN_1" := FALSE;
               //"PLC_LED_GREEN_2" := FALSE;
               //"PLC_LED_ORANGE_1" := FALSE;
               //"PLC_LED_ORANGE_2" := FALSE;
               //"PLC_LED_GREEN_CH" := FALSE;
               //"PLC_LED_RED_1" := TRUE;
               //"PLC_LED_RED_2" := TRUE;
               //"PLC_LED_RED_CH" := TRUE;

           2:  // Statement section case S2
               // GREEN = FALSE, RED = TRUE, YELLOW = TRUE
               // PED: RED = TRUE, GREEN = FALSE

               "DB_ProcessData".crossroad_output.trafficLightEast_green := FALSE;
               "DB_ProcessData".crossroad_output.trafficLightEast_red := TRUE;
               "DB_ProcessData".crossroad_output.trafficLightEast_yellow := TRUE;

               "DB_ProcessData".crossroad_output.trafficLightNorth_green := FALSE;
               "DB_ProcessData".crossroad_output.trafficLightNorth_red := TRUE;
               "DB_ProcessData".crossroad_output.trafficLightNorth_yellow := FALSE;

               "DB_ProcessData".crossroad_output.trafficLightSouth_green := FALSE;
               "DB_ProcessData".crossroad_output.trafficLightSouth_red := TRUE;
               "DB_ProcessData".crossroad_output.trafficLightSouth_yellow := FALSE;

               "DB_ProcessData".crossroad_output.trafficLightWest_green := FALSE;
               "DB_ProcessData".crossroad_output.trafficLightWest_red := TRUE;
               "DB_ProcessData".crossroad_output.trafficLightWest_yellow := TRUE;

               "DB_ProcessData".crossroad_output.pedestrianSouth1_green := FALSE;
               "DB_ProcessData".crossroad_output.pedestrianSouth1_red := TRUE;
               "DB_ProcessData".crossroad_output.pedestrianSouth2_green := FALSE;
               "DB_ProcessData".crossroad_output.pedestrianSouth2_red := TRUE;

               "DB_ProcessData".crossroad_output.pedestrianWest1_green := FALSE;
               "DB_ProcessData".crossroad_output.pedestrianWest1_red := TRUE;
               "DB_ProcessData".crossroad_output.pedestrianWest2_green := FALSE;
               "DB_ProcessData".crossroad_output.pedestrianWest2_red := TRUE;

               //"PLC_LED_GREEN_1" := FALSE;
               //"PLC_LED_GREEN_2" := FALSE;
               //"PLC_LED_ORANGE_1" := TRUE;
               //"PLC_LED_ORANGE_2" := FALSE;
               //"PLC_LED_GREEN_CH" := FALSE;
               //"PLC_LED_RED_1" := TRUE;
               //"PLC_LED_RED_2" := TRUE;
               //"PLC_LED_RED_CH" := TRUE;

           3:  // Statement section case S3
               // GREEN = TRUE, RED = FALSE, YELLOW = FALSE   // směr 1 (East, West)
               // GREEN = FALSE, RED = TRUE, YELLOW = FALSE   // směr 2 (North, South)
               // PED: RED = TRUE, GREEN = FALSE

               "DB_ProcessData".crossroad_output.trafficLightEast_green := TRUE;
               "DB_ProcessData".crossroad_output.trafficLightEast_red := FALSE;
               "DB_ProcessData".crossroad_output.trafficLightEast_yellow := FALSE;

               "DB_ProcessData".crossroad_output.trafficLightNorth_green := FALSE;
               "DB_ProcessData".crossroad_output.trafficLightNorth_red := TRUE;
               "DB_ProcessData".crossroad_output.trafficLightNorth_yellow := FALSE;

               "DB_ProcessData".crossroad_output.trafficLightSouth_green := FALSE;
               "DB_ProcessData".crossroad_output.trafficLightSouth_red := TRUE;
               "DB_ProcessData".crossroad_output.trafficLightSouth_yellow := FALSE;

               "DB_ProcessData".crossroad_output.trafficLightWest_green := TRUE;
               "DB_ProcessData".crossroad_output.trafficLightWest_red := FALSE;
               "DB_ProcessData".crossroad_output.trafficLightWest_yellow := FALSE;

               "DB_ProcessData".crossroad_output.pedestrianSouth1_green := FALSE;
               "DB_ProcessData".crossroad_output.pedestrianSouth1_red := TRUE;
               "DB_ProcessData".crossroad_output.pedestrianSouth2_green := FALSE;
               "DB_ProcessData".crossroad_output.pedestrianSouth2_red := TRUE;

               "DB_ProcessData".crossroad_output.pedestrianWest1_green := FALSE;
               "DB_ProcessData".crossroad_output.pedestrianWest1_red := TRUE;
               "DB_ProcessData".crossroad_output.pedestrianWest2_green := FALSE;
               "DB_ProcessData".crossroad_output.pedestrianWest2_red := TRUE;

               //"PLC_LED_GREEN_1" := TRUE;
               //"PLC_LED_GREEN_2" := FALSE;
               //"PLC_LED_ORANGE_1" := FALSE;
               //"PLC_LED_ORANGE_2" := FALSE;
               //"PLC_LED_GREEN_CH" := FALSE;
               //"PLC_LED_RED_1" := FALSE;
               //"PLC_LED_RED_2" := TRUE;
               //"PLC_LED_RED_CH" := TRUE;

           4:  // Statement section case S4
               // GREEN = FALSE, RED = FALSE, YELLOW = TRUE   // směr 1 (East, West)
               // GREEN = FALSE, RED = TRUE, YELLOW = FALSE   // směr 2 (North, South)
               // PED: RED = TRUE, GREEN = FALSE

               "DB_ProcessData".crossroad_output.trafficLightEast_green := FALSE;
               "DB_ProcessData".crossroad_output.trafficLightEast_red := FALSE;
               "DB_ProcessData".crossroad_output.trafficLightEast_yellow := TRUE;

               "DB_ProcessData".crossroad_output.trafficLightNorth_green := FALSE;
               "DB_ProcessData".crossroad_output.trafficLightNorth_red := TRUE;
               "DB_ProcessData".crossroad_output.trafficLightNorth_yellow := FALSE;

               "DB_ProcessData".crossroad_output.trafficLightSouth_green := FALSE;
               "DB_ProcessData".crossroad_output.trafficLightSouth_red := TRUE;
               "DB_ProcessData".crossroad_output.trafficLightSouth_yellow := FALSE;

               "DB_ProcessData".crossroad_output.trafficLightWest_green := FALSE;
               "DB_ProcessData".crossroad_output.trafficLightWest_red := FALSE;
               "DB_ProcessData".crossroad_output.trafficLightWest_yellow := TRUE;

               "DB_ProcessData".crossroad_output.pedestrianSouth1_green := FALSE;
               "DB_ProcessData".crossroad_output.pedestrianSouth1_red := TRUE;
               "DB_ProcessData".crossroad_output.pedestrianSouth2_green := FALSE;
               "DB_ProcessData".crossroad_output.pedestrianSouth2_red := TRUE;

               "DB_ProcessData".crossroad_output.pedestrianWest1_green := FALSE;
               "DB_ProcessData".crossroad_output.pedestrianWest1_red := TRUE;
               "DB_ProcessData".crossroad_output.pedestrianWest2_green := FALSE;
               "DB_ProcessData".crossroad_output.pedestrianWest2_red := TRUE;

               //"PLC_LED_GREEN_1" := FALSE;
               //"PLC_LED_GREEN_2" := FALSE;
               //"PLC_LED_ORANGE_1" := TRUE;
               //"PLC_LED_ORANGE_2" := FALSE;
               //"PLC_LED_GREEN_CH" := FALSE;
               //"PLC_LED_RED_1" := FALSE;
               //"PLC_LED_RED_2" := TRUE;
               //"PLC_LED_RED_CH" := TRUE;

           5:  // Statement section case S5
               // GREEN = FALSE, YELLOW = FALSE, RED = TRUE
               // PED: RED = TRUE, GREEN = FALSE

               "DB_ProcessData".crossroad_output.trafficLightEast_green := FALSE;
               "DB_ProcessData".crossroad_output.trafficLightEast_red := TRUE;
               "DB_ProcessData".crossroad_output.trafficLightEast_yellow := FALSE;

               "DB_ProcessData".crossroad_output.trafficLightNorth_green := FALSE;
               "DB_ProcessData".crossroad_output.trafficLightNorth_red := TRUE;
               "DB_ProcessData".crossroad_output.trafficLightNorth_yellow := FALSE;

               "DB_ProcessData".crossroad_output.trafficLightSouth_green := FALSE;
               "DB_ProcessData".crossroad_output.trafficLightSouth_red := TRUE;
               "DB_ProcessData".crossroad_output.trafficLightSouth_yellow := FALSE;

               "DB_ProcessData".crossroad_output.trafficLightWest_green := FALSE;
               "DB_ProcessData".crossroad_output.trafficLightWest_red := TRUE;
               "DB_ProcessData".crossroad_output.trafficLightWest_yellow := FALSE;

               "DB_ProcessData".crossroad_output.pedestrianSouth1_green := FALSE;
               "DB_ProcessData".crossroad_output.pedestrianSouth1_red := TRUE;
               "DB_ProcessData".crossroad_output.pedestrianSouth2_green := FALSE;
               "DB_ProcessData".crossroad_output.pedestrianSouth2_red := TRUE;

               "DB_ProcessData".crossroad_output.pedestrianWest1_green := FALSE;
               "DB_ProcessData".crossroad_output.pedestrianWest1_red := TRUE;
               "DB_ProcessData".crossroad_output.pedestrianWest2_green := FALSE;
               "DB_ProcessData".crossroad_output.pedestrianWest2_red := TRUE;

               //"PLC_LED_GREEN_1" := FALSE;
               //"PLC_LED_GREEN_2" := FALSE;
               //"PLC_LED_ORANGE_1" := FALSE;
               //"PLC_LED_ORANGE_2" := FALSE;
               //"PLC_LED_GREEN_CH" := FALSE;
               //"PLC_LED_RED_1" := TRUE;
               //"PLC_LED_RED_2" := TRUE;
               //"PLC_LED_RED_CH" := TRUE;

           6:  // Statement section case S6
               // GREEN = FALSE, RED = TRUE, YELLOW = FALSE   // směr 1 (East, West)
               // GREEN = FALSE, RED = TRUE, YELLOW = TRUE    // směr 2 (North, South)
               // PED: RED = TRUE, GREEN = FALSE (pokud není Crossroad_Walk_EN)

               "DB_ProcessData".crossroad_output.trafficLightEast_green := FALSE;
               "DB_ProcessData".crossroad_output.trafficLightEast_red := TRUE;
               "DB_ProcessData".crossroad_output.trafficLightEast_yellow := FALSE;

               "DB_ProcessData".crossroad_output.trafficLightNorth_green := FALSE;
               "DB_ProcessData".crossroad_output.trafficLightNorth_red := TRUE;
               "DB_ProcessData".crossroad_output.trafficLightNorth_yellow := TRUE;

               "DB_ProcessData".crossroad_output.trafficLightSouth_green := FALSE;
               "DB_ProcessData".crossroad_output.trafficLightSouth_red := TRUE;
               "DB_ProcessData".crossroad_output.trafficLightSouth_yellow := TRUE;

               "DB_ProcessData".crossroad_output.trafficLightWest_green := FALSE;
               "DB_ProcessData".crossroad_output.trafficLightWest_red := TRUE;
               "DB_ProcessData".crossroad_output.trafficLightWest_yellow := FALSE;

               "DB_ProcessData".crossroad_output.pedestrianSouth1_green := FALSE;
               "DB_ProcessData".crossroad_output.pedestrianSouth1_red := TRUE;
               "DB_ProcessData".crossroad_output.pedestrianSouth2_green := FALSE;
               "DB_ProcessData".crossroad_output.pedestrianSouth2_red := TRUE;

               "DB_ProcessData".crossroad_output.pedestrianWest1_green := FALSE;
               "DB_ProcessData".crossroad_output.pedestrianWest1_red := TRUE;
               "DB_ProcessData".crossroad_output.pedestrianWest2_green := FALSE;
               "DB_ProcessData".crossroad_output.pedestrianWest2_red := TRUE;

               //"PLC_LED_GREEN_1" := FALSE;
               //"PLC_LED_GREEN_2" := FALSE;
               //"PLC_LED_ORANGE_1" := FALSE;
               //"PLC_LED_ORANGE_2" := TRUE;
               //"PLC_LED_GREEN_CH" := FALSE;
               //"PLC_LED_RED_1" := TRUE;
               //"PLC_LED_RED_2" := TRUE;

               //"PLC_LED_GREEN_CH" := FALSE;
               //"PLC_LED_RED_CH" := TRUE;

               IF "Crossroad_Walk_EN" THEN
                   "DB_ProcessData".crossroad_output.pedestrianSouth1_green := TRUE;
                   "DB_ProcessData".crossroad_output.pedestrianSouth1_red := FALSE;
                   "DB_ProcessData".crossroad_output.pedestrianSouth2_green := TRUE;
                   "DB_ProcessData".crossroad_output.pedestrianSouth2_red := FALSE;

                   "DB_ProcessData".crossroad_output.pedestrianWest1_green := TRUE;
                   "DB_ProcessData".crossroad_output.pedestrianWest1_red := FALSE;
                   "DB_ProcessData".crossroad_output.pedestrianWest2_green := TRUE;
                   "DB_ProcessData".crossroad_output.pedestrianWest2_red := FALSE;

                   //"PLC_LED_GREEN_CH" := TRUE;
                   //"PLC_LED_RED_CH" := FALSE;
               END_IF;

           7:  // Statement section case S7
               // GREEN = FALSE, RED = TRUE, YELLOW = FALSE   // směr 1 (East, West)
               // GREEN = TRUE, RED = FALSE, YELLOW = FALSE   // směr 2 (North, South)
               // PED: RED = TRUE, GREEN = FALSE (pokud není Crossroad_Walk_EN)

               "DB_ProcessData".crossroad_output.trafficLightEast_green := FALSE;
               "DB_ProcessData".crossroad_output.trafficLightEast_red := TRUE;
               "DB_ProcessData".crossroad_output.trafficLightEast_yellow := FALSE;

               "DB_ProcessData".crossroad_output.trafficLightNorth_green := TRUE;
               "DB_ProcessData".crossroad_output.trafficLightNorth_red := FALSE;
               "DB_ProcessData".crossroad_output.trafficLightNorth_yellow := FALSE;

               "DB_ProcessData".crossroad_output.trafficLightSouth_green := TRUE;
               "DB_ProcessData".crossroad_output.trafficLightSouth_red := FALSE;
               "DB_ProcessData".crossroad_output.trafficLightSouth_yellow := FALSE;

               "DB_ProcessData".crossroad_output.trafficLightWest_green := FALSE;
               "DB_ProcessData".crossroad_output.trafficLightWest_red := TRUE;
               "DB_ProcessData".crossroad_output.trafficLightWest_yellow := FALSE;

               "DB_ProcessData".crossroad_output.pedestrianSouth1_green := FALSE;
               "DB_ProcessData".crossroad_output.pedestrianSouth1_red := TRUE;
               "DB_ProcessData".crossroad_output.pedestrianSouth2_green := FALSE;
               "DB_ProcessData".crossroad_output.pedestrianSouth2_red := TRUE;

               "DB_ProcessData".crossroad_output.pedestrianWest1_green := FALSE;
               "DB_ProcessData".crossroad_output.pedestrianWest1_red := TRUE;
               "DB_ProcessData".crossroad_output.pedestrianWest2_green := FALSE;
               "DB_ProcessData".crossroad_output.pedestrianWest2_red := TRUE;

               //"PLC_LED_GREEN_1" := FALSE;
               //"PLC_LED_GREEN_2" := TRUE;
               //"PLC_LED_ORANGE_1" := FALSE;
               //"PLC_LED_ORANGE_2" := FALSE;
               //"PLC_LED_RED_1" := TRUE;
               //"PLC_LED_RED_2" := FALSE;

               //"PLC_LED_GREEN_CH" := FALSE;
               //"PLC_LED_RED_CH" := TRUE;

               IF "Crossroad_Walk_EN" THEN
                   "DB_ProcessData".crossroad_output.pedestrianSouth1_green := TRUE;
                   "DB_ProcessData".crossroad_output.pedestrianSouth1_red := FALSE;
                   "DB_ProcessData".crossroad_output.pedestrianSouth2_green := TRUE;
                   "DB_ProcessData".crossroad_output.pedestrianSouth2_red := FALSE;

                   "DB_ProcessData".crossroad_output.pedestrianWest1_green := TRUE;
                   "DB_ProcessData".crossroad_output.pedestrianWest1_red := FALSE;
                   "DB_ProcessData".crossroad_output.pedestrianWest2_green := TRUE;
                   "DB_ProcessData".crossroad_output.pedestrianWest2_red := FALSE;

                   //"PLC_LED_GREEN_CH" := TRUE;
                   //"PLC_LED_RED_CH" := FALSE;
               END_IF;

           8:  // Statement section case S8
               // GREEN = FALSE, RED = TRUE, YELLOW = FALSE   // směr 1 (East, West)
               // GREEN = FALSE, RED = FALSE, YELLOW = TRUE   // směr 2 (North, South)
               // PED: RED = TRUE, GREEN = FALSE

               "DB_ProcessData".crossroad_output.trafficLightEast_green := FALSE;
               "DB_ProcessData".crossroad_output.trafficLightEast_red := TRUE;
               "DB_ProcessData".crossroad_output.trafficLightEast_yellow := FALSE;

               "DB_ProcessData".crossroad_output.trafficLightNorth_green := FALSE;
               "DB_ProcessData".crossroad_output.trafficLightNorth_red := FALSE;
               "DB_ProcessData".crossroad_output.trafficLightNorth_yellow := TRUE;

               "DB_ProcessData".crossroad_output.trafficLightSouth_green := FALSE;
               "DB_ProcessData".crossroad_output.trafficLightSouth_red := FALSE;
               "DB_ProcessData".crossroad_output.trafficLightSouth_yellow := TRUE;

               "DB_ProcessData".crossroad_output.trafficLightWest_green := FALSE;
               "DB_ProcessData".crossroad_output.trafficLightWest_red := TRUE;
               "DB_ProcessData".crossroad_output.trafficLightWest_yellow := FALSE;

               "DB_ProcessData".crossroad_output.pedestrianSouth1_green := FALSE;
               "DB_ProcessData".crossroad_output.pedestrianSouth1_red := TRUE;
               "DB_ProcessData".crossroad_output.pedestrianSouth2_green := FALSE;
               "DB_ProcessData".crossroad_output.pedestrianSouth2_red := TRUE;

               "DB_ProcessData".crossroad_output.pedestrianWest1_green := FALSE;
               "DB_ProcessData".crossroad_output.pedestrianWest1_red := TRUE;
               "DB_ProcessData".crossroad_output.pedestrianWest2_green := FALSE;
               "DB_ProcessData".crossroad_output.pedestrianWest2_red := TRUE;

               //"PLC_LED_GREEN_1" := FALSE;
               //"PLC_LED_GREEN_2" := FALSE;
               //"PLC_LED_ORANGE_1" := FALSE;
               //"PLC_LED_ORANGE_2" := TRUE;
               //"PLC_LED_GREEN_CH" := FALSE;
               //"PLC_LED_RED_1" := TRUE;
               //"PLC_LED_RED_2" := FALSE;
               //"PLC_LED_RED_CH" := TRUE;

           9:  // Statement section case S9
               // GREEN = FALSE, YELLOW = FALSE, RED = TRUE
               // PED: RED = TRUE, GREEN = FALSE

               "DB_ProcessData".crossroad_output.trafficLightEast_green := FALSE;
               "DB_ProcessData".crossroad_output.trafficLightEast_red := TRUE;
               "DB_ProcessData".crossroad_output.trafficLightEast_yellow := FALSE;

               "DB_ProcessData".crossroad_output.trafficLightNorth_green := FALSE;
               "DB_ProcessData".crossroad_output.trafficLightNorth_red := TRUE;
               "DB_ProcessData".crossroad_output.trafficLightNorth_yellow := FALSE;

               "DB_ProcessData".crossroad_output.trafficLightSouth_green := FALSE;
               "DB_ProcessData".crossroad_output.trafficLightSouth_red := TRUE;
               "DB_ProcessData".crossroad_output.trafficLightSouth_yellow := FALSE;

               "DB_ProcessData".crossroad_output.trafficLightWest_green := FALSE;
               "DB_ProcessData".crossroad_output.trafficLightWest_red := TRUE;
               "DB_ProcessData".crossroad_output.trafficLightWest_yellow := FALSE;

               "DB_ProcessData".crossroad_output.pedestrianSouth1_green := FALSE;
               "DB_ProcessData".crossroad_output.pedestrianSouth1_red := TRUE;
               "DB_ProcessData".crossroad_output.pedestrianSouth2_green := FALSE;
               "DB_ProcessData".crossroad_output.pedestrianSouth2_red := TRUE;

               "DB_ProcessData".crossroad_output.pedestrianWest1_green := FALSE;
               "DB_ProcessData".crossroad_output.pedestrianWest1_red := TRUE;
               "DB_ProcessData".crossroad_output.pedestrianWest2_green := FALSE;
               "DB_ProcessData".crossroad_output.pedestrianWest2_red := TRUE;

               //"PLC_LED_GREEN_1" := FALSE;
               //"PLC_LED_GREEN_2" := FALSE;
               //"PLC_LED_ORANGE_1" := FALSE;
               //"PLC_LED_ORANGE_2" := FALSE;
               //"PLC_LED_GREEN_CH" := FALSE;
               //"PLC_LED_RED_1" := TRUE;
               //"PLC_LED_RED_2" := TRUE;
               //"PLC_LED_RED_CH" := TRUE;

               "Crossroad_Walk_EN" := FALSE;

           ELSE  // Statement section ELSE
               "DB_ProcessData".crossroad_output.trafficLightEast_green := FALSE;
               "DB_ProcessData".crossroad_output.trafficLightEast_red := FALSE;
               "DB_ProcessData".crossroad_output.trafficLightEast_yellow := FALSE;

               "DB_ProcessData".crossroad_output.trafficLightNorth_green := FALSE;
               "DB_ProcessData".crossroad_output.trafficLightNorth_red := FALSE;
               "DB_ProcessData".crossroad_output.trafficLightNorth_yellow := FALSE;

               "DB_ProcessData".crossroad_output.trafficLightSouth_green := FALSE;
               "DB_ProcessData".crossroad_output.trafficLightSouth_red := FALSE;
               "DB_ProcessData".crossroad_output.trafficLightSouth_yellow := FALSE;

               "DB_ProcessData".crossroad_output.trafficLightWest_green := FALSE;
               "DB_ProcessData".crossroad_output.trafficLightWest_red := FALSE;
               "DB_ProcessData".crossroad_output.trafficLightWest_yellow := FALSE;

               "DB_ProcessData".crossroad_output.pedestrianSouth1_green := FALSE;
               "DB_ProcessData".crossroad_output.pedestrianSouth1_red := FALSE;
               "DB_ProcessData".crossroad_output.pedestrianSouth2_green := FALSE;
               "DB_ProcessData".crossroad_output.pedestrianSouth2_red := FALSE;

               "DB_ProcessData".crossroad_output.pedestrianWest1_green := FALSE;
               "DB_ProcessData".crossroad_output.pedestrianWest1_red := FALSE;
               "DB_ProcessData".crossroad_output.pedestrianWest2_green := FALSE;
               "DB_ProcessData".crossroad_output.pedestrianWest2_red := FALSE;

               //"PLC_LED_GREEN_1" := FALSE;
               //"PLC_LED_GREEN_2" := FALSE;
               //"PLC_LED_ORANGE_1" := FALSE;
               //"PLC_LED_ORANGE_2" := FALSE;
               //"PLC_LED_RED_1" := FALSE;
               //"PLC_LED_RED_2" := FALSE;
               //"PLC_LED_GREEN_CH" := FALSE;
               //"PLC_LED_RED_CH" := FALSE;

               "Crossroad_Walk_EN" := FALSE;
       END_CASE;
   END_IF;
END_REGION

REGION Network 6 (SCL): Pedestrians bnts
   IF "DB_ProcessData".crossroad_input.btnSouthCrosswalk1 OR "DB_ProcessData".crossroad_input.btnSouthCrosswalk2 OR "DB_ProcessData".crossroad_input.btnWestCrosswalk1 OR "DB_ProcessData".crossroad_input.btnWestCrosswalk2 THEN
       "Crossroad_Walk_EN" := TRUE;
   END_IF;
END_REGION
END_FUNCTION

// folder: Crosswalk

FUNCTION "Crosswalk_MAIN" : Void   // FC1, LAD
{ S7_Optimized_Access := 'TRUE' }
VERSION : 0.1
BEGIN

REGION Network 1: Control
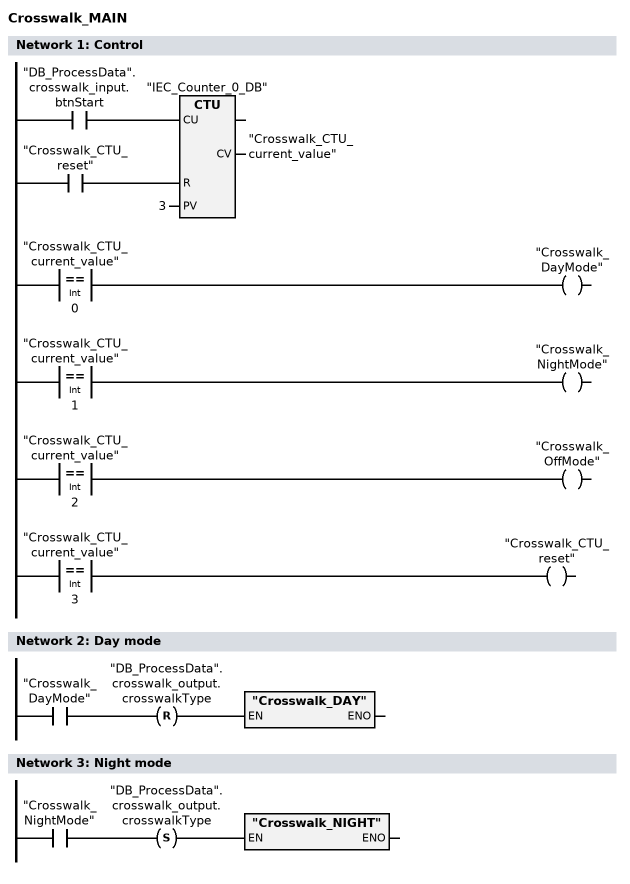
   "IEC_Counter_0_DB".CTU(CU := "DB_ProcessData".crosswalk_input.btnStart,
                          R := "Crosswalk_CTU_reset",
                          PV := 3,
                          CV => "Crosswalk_CTU_current_value");
   "Crosswalk_DayMode" := "Crosswalk_CTU_current_value" = 0;
   "Crosswalk_NightMode" := "Crosswalk_CTU_current_value" = 1;
   "Crosswalk_OffMode" := "Crosswalk_CTU_current_value" = 2;
   "Crosswalk_CTU_reset" := "Crosswalk_CTU_current_value" = 3;
END_REGION

REGION Network 2: Day mode
   RUNG wire#powerrail
      Contact( "Crosswalk_DayMode" )
      R_Coil( "DB_ProcessData".crosswalk_output.crosswalkType )
      "Crosswalk_DAY"()
   END_RUNG
   // the same network as SCL:
   IF "Crosswalk_DayMode" THEN
       "DB_ProcessData".crosswalk_output.crosswalkType := FALSE;
       "Crosswalk_DAY"();
   END_IF;
END_REGION

REGION Network 3: Night mode
   RUNG wire#powerrail
      Contact( "Crosswalk_NightMode" )
      S_Coil( "DB_ProcessData".crosswalk_output.crosswalkType )
      "Crosswalk_NIGHT"()
   END_RUNG
   // the same network as SCL:
   IF "Crosswalk_NightMode" THEN
       "DB_ProcessData".crosswalk_output.crosswalkType := TRUE;
       "Crosswalk_NIGHT"();
   END_IF;
END_REGION

REGION Network 4 (SCL): Off mode
   IF "Crosswalk_OffMode" = TRUE THEN
       "DB_ProcessData".crosswalk_output.pedestrianLightGreen1 := FALSE;
       "DB_ProcessData".crosswalk_output.pedestrianLightGreen2 := FALSE;
       "DB_ProcessData".crosswalk_output.pedestrianLightRed1 := FALSE;
       "DB_ProcessData".crosswalk_output.pedestrianLightRed2 := FALSE;
       "DB_ProcessData".crosswalk_output.trafficLightGreen1 := FALSE;
       "DB_ProcessData".crosswalk_output.trafficLightGreen2 := FALSE;
       "DB_ProcessData".crosswalk_output.trafficLightsRed1 := FALSE;
       "DB_ProcessData".crosswalk_output.trafficLightsRed2 := FALSE;
       "DB_ProcessData".crosswalk_output.trafficLightsYellow1 := FALSE;
       "DB_ProcessData".crosswalk_output.trafficLightsYellow2 := FALSE;
   END_IF;
END_REGION
END_FUNCTION

FUNCTION "Crosswalk_DAY" : Void   // FC2, LAD
{ S7_Optimized_Access := 'TRUE' }
VERSION : 0.1
   VAR_TEMP   // added for the SCL form of the ladder/FBD networks
      _w1 : Bool;
   END_VAR
BEGIN

REGION Network 1: Green
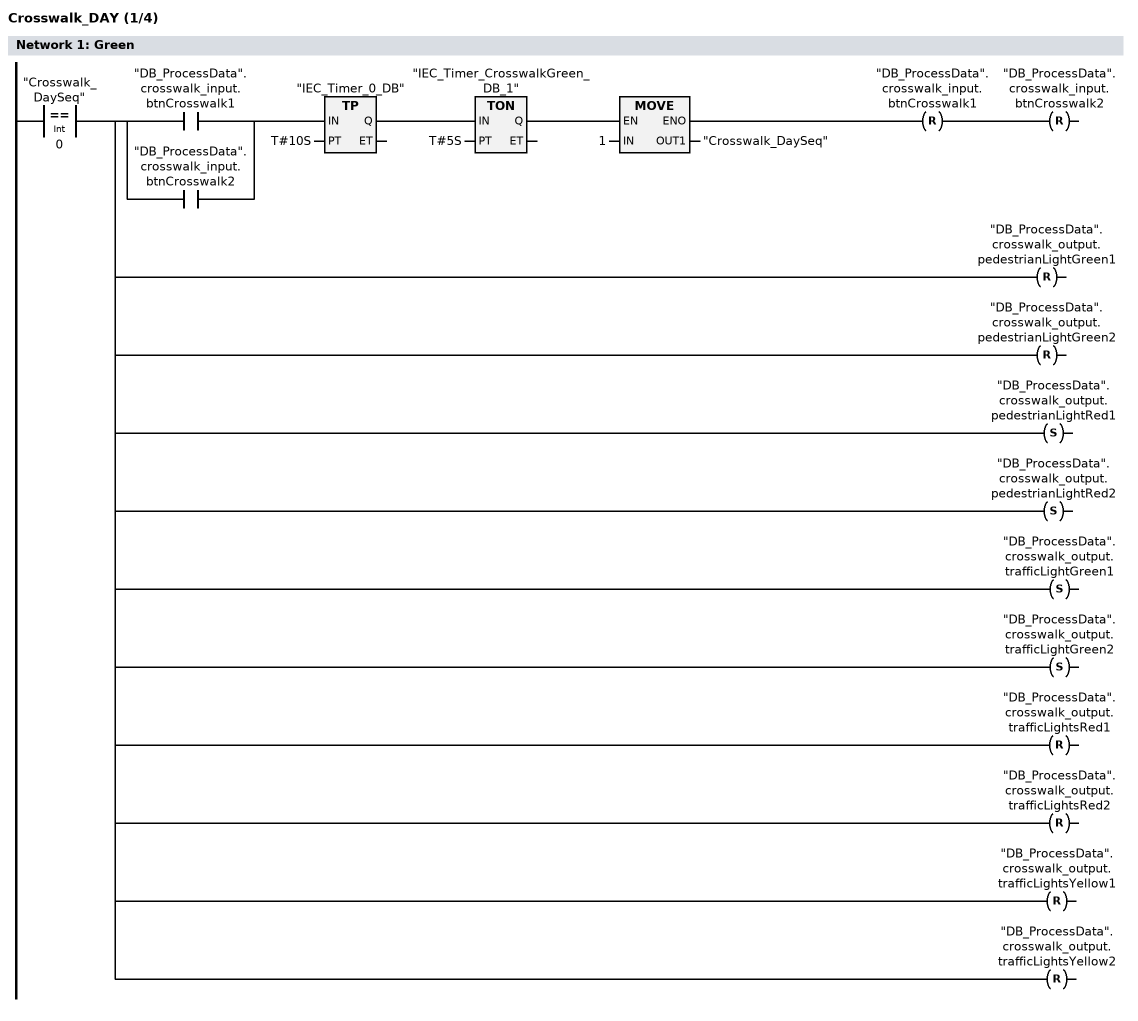
   #_w1 := "Crosswalk_DaySeq" = 0;
   "IEC_Timer_0_DB".TP(IN := #_w1 AND ("DB_ProcessData".crosswalk_input.btnCrosswalk1 OR "DB_ProcessData".crosswalk_input.btnCrosswalk2),
                       PT := T#10S);
   "IEC_Timer_CrosswalkGreen_DB_1".TON(IN := "IEC_Timer_0_DB".Q, PT := T#5S);
   IF "IEC_Timer_CrosswalkGreen_DB_1".Q THEN
       "Crosswalk_DaySeq" := 1;
       "DB_ProcessData".crosswalk_input.btnCrosswalk1 := FALSE;
       "DB_ProcessData".crosswalk_input.btnCrosswalk2 := FALSE;
   END_IF;
   IF #_w1 THEN
       "DB_ProcessData".crosswalk_output.pedestrianLightGreen1 := FALSE;
       "DB_ProcessData".crosswalk_output.pedestrianLightGreen2 := FALSE;
       "DB_ProcessData".crosswalk_output.pedestrianLightRed1 := TRUE;
       "DB_ProcessData".crosswalk_output.pedestrianLightRed2 := TRUE;
       "DB_ProcessData".crosswalk_output.trafficLightGreen1 := TRUE;
       "DB_ProcessData".crosswalk_output.trafficLightGreen2 := TRUE;
       "DB_ProcessData".crosswalk_output.trafficLightsRed1 := FALSE;
       "DB_ProcessData".crosswalk_output.trafficLightsRed2 := FALSE;
       "DB_ProcessData".crosswalk_output.trafficLightsYellow1 := FALSE;
       "DB_ProcessData".crosswalk_output.trafficLightsYellow2 := FALSE;
   END_IF;
END_REGION

REGION Network 2: Yellow1
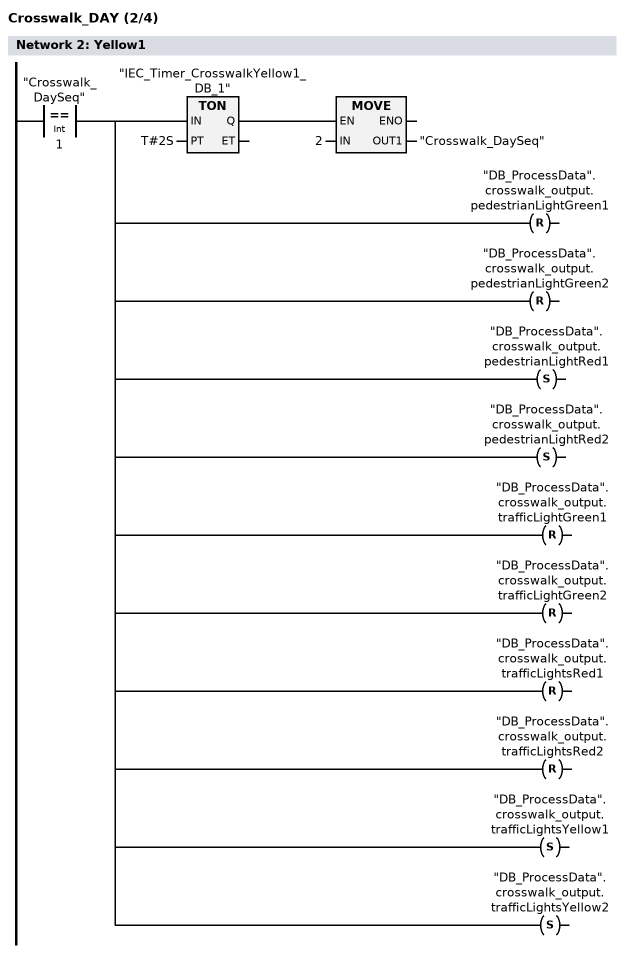
   #_w1 := "Crosswalk_DaySeq" = 1;
   "IEC_Timer_CrosswalkYellow1_DB_1".TON(IN := #_w1, PT := T#2S);
   IF "IEC_Timer_CrosswalkYellow1_DB_1".Q THEN "Crosswalk_DaySeq" := 2; END_IF;
   IF #_w1 THEN
       "DB_ProcessData".crosswalk_output.pedestrianLightGreen1 := FALSE;
       "DB_ProcessData".crosswalk_output.pedestrianLightGreen2 := FALSE;
       "DB_ProcessData".crosswalk_output.pedestrianLightRed1 := TRUE;
       "DB_ProcessData".crosswalk_output.pedestrianLightRed2 := TRUE;
       "DB_ProcessData".crosswalk_output.trafficLightGreen1 := FALSE;
       "DB_ProcessData".crosswalk_output.trafficLightGreen2 := FALSE;
       "DB_ProcessData".crosswalk_output.trafficLightsRed1 := FALSE;
       "DB_ProcessData".crosswalk_output.trafficLightsRed2 := FALSE;
       "DB_ProcessData".crosswalk_output.trafficLightsYellow1 := TRUE;
       "DB_ProcessData".crosswalk_output.trafficLightsYellow2 := TRUE;
   END_IF;
END_REGION

REGION Network 3: Red
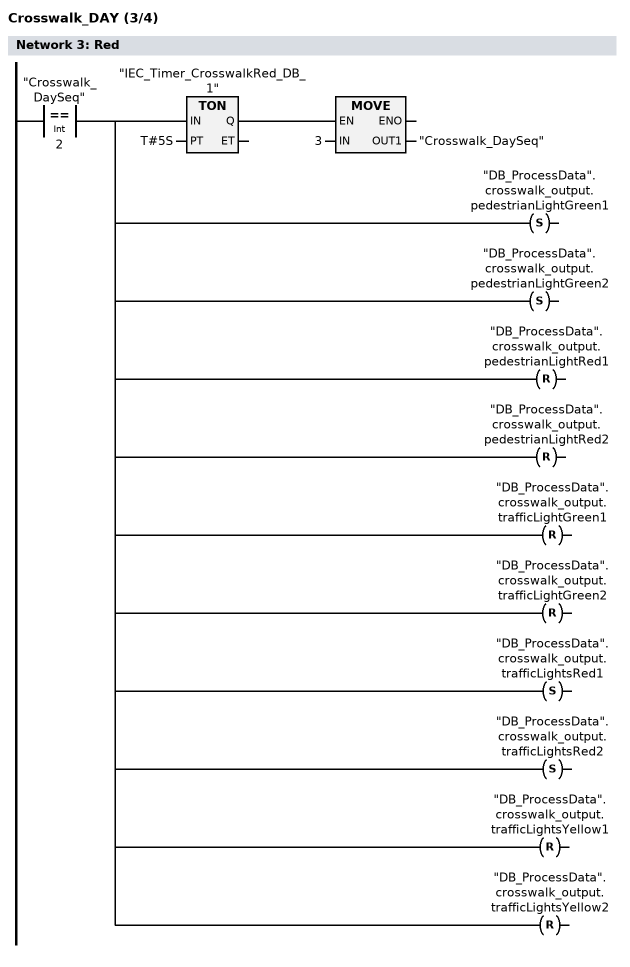
   #_w1 := "Crosswalk_DaySeq" = 2;
   "IEC_Timer_CrosswalkRed_DB_1".TON(IN := #_w1, PT := T#5S);
   IF "IEC_Timer_CrosswalkRed_DB_1".Q THEN "Crosswalk_DaySeq" := 3; END_IF;
   IF #_w1 THEN
       "DB_ProcessData".crosswalk_output.pedestrianLightGreen1 := TRUE;
       "DB_ProcessData".crosswalk_output.pedestrianLightGreen2 := TRUE;
       "DB_ProcessData".crosswalk_output.pedestrianLightRed1 := FALSE;
       "DB_ProcessData".crosswalk_output.pedestrianLightRed2 := FALSE;
       "DB_ProcessData".crosswalk_output.trafficLightGreen1 := FALSE;
       "DB_ProcessData".crosswalk_output.trafficLightGreen2 := FALSE;
       "DB_ProcessData".crosswalk_output.trafficLightsRed1 := TRUE;
       "DB_ProcessData".crosswalk_output.trafficLightsRed2 := TRUE;
       "DB_ProcessData".crosswalk_output.trafficLightsYellow1 := FALSE;
       "DB_ProcessData".crosswalk_output.trafficLightsYellow2 := FALSE;
   END_IF;
END_REGION

REGION Network 4: Yellow2
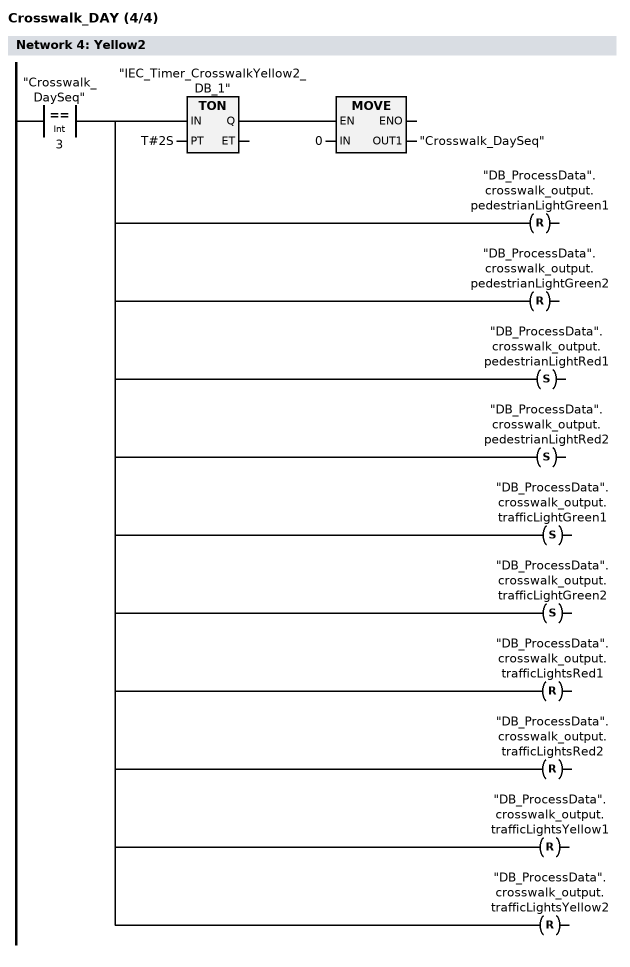
   #_w1 := "Crosswalk_DaySeq" = 3;
   "IEC_Timer_CrosswalkYellow2_DB_1".TON(IN := #_w1, PT := T#2S);
   IF "IEC_Timer_CrosswalkYellow2_DB_1".Q THEN "Crosswalk_DaySeq" := 0; END_IF;
   IF #_w1 THEN
       "DB_ProcessData".crosswalk_output.pedestrianLightGreen1 := FALSE;
       "DB_ProcessData".crosswalk_output.pedestrianLightGreen2 := FALSE;
       "DB_ProcessData".crosswalk_output.pedestrianLightRed1 := TRUE;
       "DB_ProcessData".crosswalk_output.pedestrianLightRed2 := TRUE;
       "DB_ProcessData".crosswalk_output.trafficLightGreen1 := TRUE;
       "DB_ProcessData".crosswalk_output.trafficLightGreen2 := TRUE;
       "DB_ProcessData".crosswalk_output.trafficLightsRed1 := FALSE;
       "DB_ProcessData".crosswalk_output.trafficLightsRed2 := FALSE;
       "DB_ProcessData".crosswalk_output.trafficLightsYellow1 := FALSE;
       "DB_ProcessData".crosswalk_output.trafficLightsYellow2 := FALSE;
   END_IF;
END_REGION
END_FUNCTION

FUNCTION "Crosswalk_NIGHT" : Void   // FC3, LAD
{ S7_Optimized_Access := 'TRUE' }
VERSION : 0.1
   VAR_TEMP   // added for the SCL form of the ladder/FBD networks
      _w1 : Bool;
   END_VAR
BEGIN

REGION Network 1: On
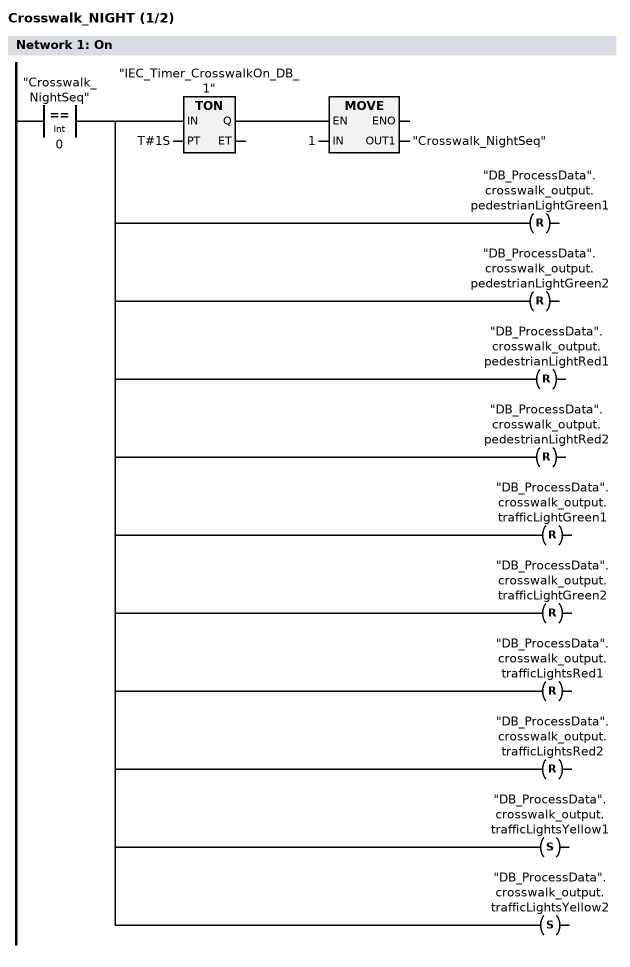
   #_w1 := "Crosswalk_NightSeq" = 0;
   "IEC_Timer_CrosswalkOn_DB_1".TON(IN := #_w1, PT := T#1S);
   IF "IEC_Timer_CrosswalkOn_DB_1".Q THEN "Crosswalk_NightSeq" := 1; END_IF;
   IF #_w1 THEN
       "DB_ProcessData".crosswalk_output.pedestrianLightGreen1 := FALSE;
       "DB_ProcessData".crosswalk_output.pedestrianLightGreen2 := FALSE;
       "DB_ProcessData".crosswalk_output.pedestrianLightRed1 := FALSE;
       "DB_ProcessData".crosswalk_output.pedestrianLightRed2 := FALSE;
       "DB_ProcessData".crosswalk_output.trafficLightGreen1 := FALSE;
       "DB_ProcessData".crosswalk_output.trafficLightGreen2 := FALSE;
       "DB_ProcessData".crosswalk_output.trafficLightsRed1 := FALSE;
       "DB_ProcessData".crosswalk_output.trafficLightsRed2 := FALSE;
       "DB_ProcessData".crosswalk_output.trafficLightsYellow1 := TRUE;
       "DB_ProcessData".crosswalk_output.trafficLightsYellow2 := TRUE;
   END_IF;
END_REGION

REGION Network 2: Off
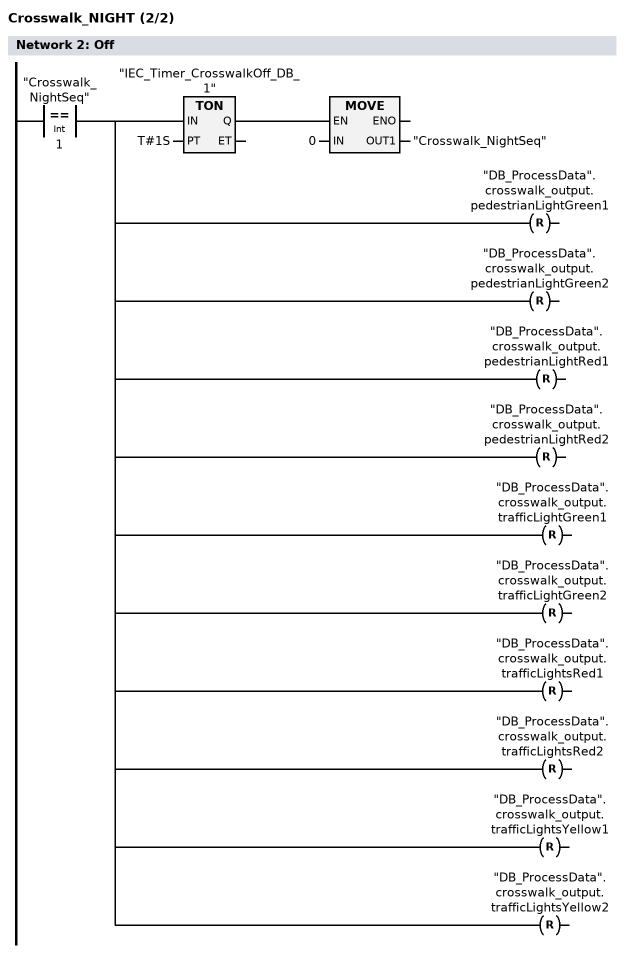
   #_w1 := "Crosswalk_NightSeq" = 1;
   "IEC_Timer_CrosswalkOff_DB_1".TON(IN := #_w1, PT := T#1S);
   IF "IEC_Timer_CrosswalkOff_DB_1".Q THEN "Crosswalk_NightSeq" := 0; END_IF;
   IF #_w1 THEN
       "DB_ProcessData".crosswalk_output.pedestrianLightGreen1 := FALSE;
       "DB_ProcessData".crosswalk_output.pedestrianLightGreen2 := FALSE;
       "DB_ProcessData".crosswalk_output.pedestrianLightRed1 := FALSE;
       "DB_ProcessData".crosswalk_output.pedestrianLightRed2 := FALSE;
       "DB_ProcessData".crosswalk_output.trafficLightGreen1 := FALSE;
       "DB_ProcessData".crosswalk_output.trafficLightGreen2 := FALSE;
       "DB_ProcessData".crosswalk_output.trafficLightsRed1 := FALSE;
       "DB_ProcessData".crosswalk_output.trafficLightsRed2 := FALSE;
       "DB_ProcessData".crosswalk_output.trafficLightsYellow1 := FALSE;
       "DB_ProcessData".crosswalk_output.trafficLightsYellow2 := FALSE;
   END_IF;
END_REGION
END_FUNCTION

// folder: Regulator

FUNCTION "Regulator_PID" : Void   // FC5, LAD
{ S7_Optimized_Access := 'TRUE' }
VERSION : 0.1
BEGIN

REGION Network 1 (SCL)
   CASE "DB_ProcessData".regulator_input.order OF
       1:
           "Regulator_PV" := "DB_ProcessData".regulator_input.Uc1;
       2:
           "Regulator_PV" := "DB_ProcessData".regulator_input.Uc2;
       ELSE
           "Regulator_PV" := 0;
   END_CASE;

   "Regulator_SetPoint" := 50;
END_REGION

REGION Network 2
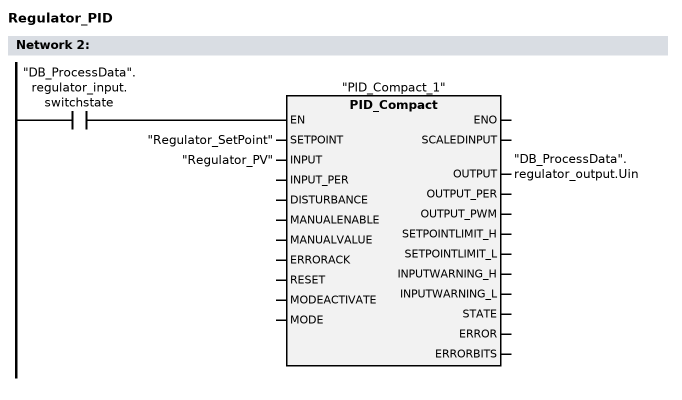
   IF "DB_ProcessData".regulator_input.switchstate THEN
       "PID_Compact_1"(Setpoint := "Regulator_SetPoint",   // PID_Compact
                       Input := "Regulator_PV",
                       Output => "DB_ProcessData".regulator_output.Uin);
   END_IF;
END_REGION
END_FUNCTION

// ===== PLC "R2D2_OPCUA"  CPU 1212C DC/DC/DC =====

VAR_GLOBAL   // PLC tag table "Default tag table"
   "Clock_Byte" AT %MB0 : Byte;
   "Clock_10Hz" AT %M0.0 : Bool;
   "Clock_5Hz" AT %M0.1 : Bool;
   "Clock_2.5Hz" AT %M0.2 : Bool;
   "Clock_2Hz" AT %M0.3 : Bool;
   "Clock_1.25Hz" AT %M0.4 : Bool;
   "Clock_1Hz" AT %M0.5 : Bool;
   "Clock_0.625Hz" AT %M0.6 : Bool;
   "Clock_0.5Hz" AT %M0.7 : Bool;
   "System_Byte" AT %MB1 : Byte;
   "FirstScan" AT %M1.0 : Bool;
   "DiagStatusUpdate" AT %M1.1 : Bool;
   "AlwaysTRUE" AT %M1.2 : Bool;
   "AlwaysFALSE" AT %M1.3 : Bool;
END_VAR

VAR_GLOBAL   // PLC tag table "Regulator"
   "Regulator_PV" AT %MD100 : Real;
   "Regulator_SetPoint" AT %MD104 : Real;
END_VAR

VAR_GLOBAL   // PLC tag table "CarLight"
   "CarLight_Tag1" AT %I0.0 : Bool;
END_VAR

VAR_GLOBAL   // PLC tag table "Crossroad"
   "Crossroad_Tag_1" AT %M300.0 : Bool;
   "Crossroad_Tag_2" AT %M300.1 : Bool;
   "Crossroad_Tag_3" AT %MW302 : Word;
   "Crossroad_MEM 0" AT %M304.0 : Bool;
   "Crossroad_MEM 1" AT %M304.1 : Bool;
   "Crossroad_MEM 2" AT %M304.2 : Bool;
   "Crossroad_MEM 3" AT %M304.3 : Bool;
   "Crossroad_MEM 5" AT %M304.4 : Bool;
   "Crossroad_MEM 6" AT %M304.5 : Bool;
   "Crossroad_Clock" AT %MW328 : Int;
   "Crossroad_DayModeState" AT %MB305 : USInt;
   "Crossroad_ActualLengthState" AT %MD316 : Time;
   "Crossorad_HoursDayStart" AT %MW320 : Int;
   "Crossroad_HoursDayEnd" AT %MW322 : Int;
   "Crossroad_DayStarts" AT %MW324 : Int;
   "Crossroad_DayEnds" AT %MW326 : Int;
   "Crossroad_S1" AT %MB306 : USInt;
   "Crossroad_S2" AT %MB307 : USInt;
   "Crossroad_S3" AT %MB308 : USInt;
   "Crossroad_S4" AT %MB309 : USInt;
   "Crossroad_S5" AT %MB310 : USInt;
   "Crossroad_S6" AT %MB311 : USInt;
   "Crossroad_S7" AT %MB312 : USInt;
   "Crossroad_S8" AT %MB313 : USInt;
   "Crossroad_S9" AT %MB314 : USInt;
   "Crossroad_Walk_EN" AT %M330.0 : Bool;
END_VAR

VAR_GLOBAL   // PLC tag table "Crosswalk"
   "Crosswalk_CTU_current_value" AT %MW200 : Int;
   "Crosswalk_CTU_reset" AT %M202.0 : Bool;
   "Crosswalk_DayMode" AT %M202.1 : Bool;
   "Crosswalk_NightMode" AT %M202.2 : Bool;
   "Crosswalk_OffMode" AT %M202.3 : Bool;
   "Crosswalk_DaySeq" AT %MW204 : Int;
   "Crosswalk_NightSeq" AT %MW206 : Int;
END_VAR

TYPE "Crossroad_Input"
   STRUCT
      btnStart : Bool := FALSE;
      btnPause : Bool := FALSE;
      btnStop : Bool := FALSE;
      btnWestCrosswalk1 : Bool := FALSE;
      btnWestCrosswalk2 : Bool := FALSE;
      btnSouthCrosswalk1 : Bool := FALSE;
      btnSouthCrosswalk2 : Bool := FALSE;
      spare1 : DWord := 0;
      spare2 : DWord := 0;
      spare3 : DWord := 0;
      spare4 : DWord := 0;
   END_STRUCT;
END_TYPE

TYPE "Crossroad_Output"
   STRUCT
      crossroadType : Bool := FALSE;
      trafficLightNorth_green : Bool := FALSE;
      trafficLightNorth_yellow : Bool := FALSE;
      trafficLightNorth_red : Bool := FALSE;
      trafficLightSouth_green : Bool := FALSE;
      trafficLightSouth_yellow : Bool := FALSE;
      trafficLightSouth_red : Bool := FALSE;
      trafficLightWest_green : Bool := FALSE;
      trafficLightWest_yellow : Bool := FALSE;
      trafficLightWest_red : Bool := FALSE;
      trafficLightEast_green : Bool := FALSE;
      trafficLightEast_yellow : Bool := FALSE;
      trafficLightEast_red : Bool := FALSE;
      pedestrianSouth1_green : Bool := FALSE;
      pedestrianSouth1_red : Bool := FALSE;
      pedestrianSouth2_green : Bool := FALSE;
      pedestrianSouth2_red : Bool := FALSE;
      pedestrianWest1_green : Bool := FALSE;
      pedestrianWest1_red : Bool := FALSE;
      pedestrianWest2_green : Bool := FALSE;
      pedestrianWest2_red : Bool := FALSE;
      spare1 : DWord := 0;
      spare2 : DWord := 0;
      spare3 : DWord := 0;
      spare4 : DWord := 0;
   END_STRUCT;
END_TYPE

TYPE "Crosswalk_Input"
   STRUCT
      btnStart : Bool := FALSE;
      btnPause : Bool := FALSE;
      btnStop : Bool := FALSE;
      btnCrosswalk1 : Bool := FALSE;
      btnCrosswalk2 : Bool := FALSE;
      spare1 : DWord := 0;
      spare2 : DWord := 0;
      spare3 : DWord := 0;
      spare4 : DWord := 0;
   END_STRUCT;
END_TYPE

TYPE "Crosswalk_Output"
   STRUCT
      crosswalkType : Bool := FALSE;
      trafficLightGreen1 : Bool := FALSE;
      trafficLightsYellow1 : Bool := FALSE;
      trafficLightsRed1 : Bool := FALSE;
      trafficLightGreen2 : Bool := FALSE;
      trafficLightsYellow2 : Bool := FALSE;
      trafficLightsRed2 : Bool := FALSE;
      pedestrianLightGreen1 : Bool := FALSE;
      pedestrianLightRed1 : Bool := FALSE;
      pedestrianLightGreen2 : Bool := FALSE;
      pedestrianLightRed2 : Bool := FALSE;
      spare1 : DWord := 0;
      spare2 : DWord := 0;
      spare3 : DWord := 0;
      spare4 : DWord := 0;
   END_STRUCT;
END_TYPE

TYPE "Regulator_Input"
   STRUCT
      btnReset : Bool := FALSE;
      switchstate : Bool := FALSE;
      order : Int := 1;
      R1 : Real := 0.0;
      R2 : Real := 0.0;
      C1 : Real := 0.0;
      C2 : Real := 0.0;
      Uc1 : Real := 0.0;
      Uc2 : Real := 0.0;
      Td : Real := 0.0;
      Ts : Real := 0.0;
      spare1 : DWord := 0;
      spare2 : DWord := 0;
      spare3 : DWord := 0;
      spare4 : DWord := 0;
   END_STRUCT;
END_TYPE

TYPE "Regulator_Output"
   STRUCT
      Uin : Real := 0.0;
      spare1 : DWord := 0;
      spare2 : DWord := 0;
      spare3 : DWord := 0;
      spare4 : DWord := 0;
   END_STRUCT;
END_TYPE

TYPE "CarLight_Input"
   STRUCT
      btnReset : Bool := FALSE;
      error : Bool := FALSE;
      sensorLight : Bool := FALSE;
      sensorConnectorConnected : Bool := FALSE;
      result : Bool := FALSE;
      spare1 : DWord := 0;
      spare2 : DWord := 0;
      spare3 : DWord := 0;
      spare4 : DWord := 0;
   END_STRUCT;
END_TYPE

TYPE "CarLight_Output"
   STRUCT
      lowBeamLight : Bool := FALSE;
      highBeamLight : Bool := FALSE;
      turnLight : Bool := FALSE;
      spare1 : DWord := 0;
      spare2 : DWord := 0;
      spare3 : DWord := 0;
      spare4 : DWord := 0;
   END_STRUCT;
END_TYPE

DATA_BLOCK "DB_ProcessData"   // DB1
{ S7_Optimized_Access := 'TRUE' }
VERSION : 0.1
   VAR
      crossroad_input : "Crossroad_Input";
      crossroad_output : "Crossroad_Output";
      crosswalk_input : "Crosswalk_Input";
      crosswalk_output : "Crosswalk_Output";
      regulator_input : "Regulator_Input";
      regulator_output : "Regulator_Output";
      carlight_input : "CarLight_Input";
      carlight_output : "CarLight_Output";
   END_VAR
BEGIN
END_DATA_BLOCK

// folder: CarLight

DATA_BLOCK "CarLight_SCL_DB"   // DB12
{ S7_Optimized_Access := 'TRUE' }
VERSION : 0.1
// stored: InstanceOfName CarLight_SCL
"CarLight_SCL"
BEGIN
END_DATA_BLOCK

// folder: System blocks/Program resources

DATA_BLOCK "IEC_Counter_0_DB"   // DB2
{ S7_Optimized_Access := 'TRUE' }
AUTHOR : Simatic
FAMILY : IEC
NAME : CNTR
VERSION : 1.0
// stored: InstanceOfName IEC_COUNTER
"IEC_COUNTER"
BEGIN
END_DATA_BLOCK

DATA_BLOCK "IEC_Timer_0_DB"   // DB3
{ S7_Optimized_Access := 'TRUE' }
AUTHOR : Simatic
FAMILY : IEC
NAME : IEC_TMR
VERSION : 1.0
// stored: InstanceOfName IEC_TIMER
"IEC_TIMER"
BEGIN
END_DATA_BLOCK

DATA_BLOCK "IEC_Timer_CrosswalkGreen_DB_1"   // DB4
{ S7_Optimized_Access := 'TRUE' }
AUTHOR : Simatic
FAMILY : IEC
NAME : IEC_TMR
VERSION : 1.0
// stored: InstanceOfName IEC_TIMER
"IEC_TIMER"
BEGIN
END_DATA_BLOCK

DATA_BLOCK "IEC_Timer_CrosswalkYellow1_DB_1"   // DB5
{ S7_Optimized_Access := 'TRUE' }
AUTHOR : Simatic
FAMILY : IEC
NAME : IEC_TMR
VERSION : 1.0
// stored: InstanceOfName IEC_TIMER
"IEC_TIMER"
BEGIN
END_DATA_BLOCK

DATA_BLOCK "IEC_Timer_CrosswalkRed_DB_1"   // DB6
{ S7_Optimized_Access := 'TRUE' }
AUTHOR : Simatic
FAMILY : IEC
NAME : IEC_TMR
VERSION : 1.0
// stored: InstanceOfName IEC_TIMER
"IEC_TIMER"
BEGIN
END_DATA_BLOCK

DATA_BLOCK "IEC_Timer_CrosswalkYellow2_DB_1"   // DB7
{ S7_Optimized_Access := 'TRUE' }
AUTHOR : Simatic
FAMILY : IEC
NAME : IEC_TMR
VERSION : 1.0
// stored: InstanceOfName IEC_TIMER
"IEC_TIMER"
BEGIN
END_DATA_BLOCK

DATA_BLOCK "IEC_Timer_CrosswalkOn_DB_1"   // DB8
{ S7_Optimized_Access := 'TRUE' }
AUTHOR : Simatic
FAMILY : IEC
NAME : IEC_TMR
VERSION : 1.0
// stored: InstanceOfName IEC_TIMER
"IEC_TIMER"
BEGIN
END_DATA_BLOCK

DATA_BLOCK "IEC_Timer_CrosswalkOff_DB_1"   // DB9
{ S7_Optimized_Access := 'TRUE' }
AUTHOR : Simatic
FAMILY : IEC
NAME : IEC_TMR
VERSION : 1.0
// stored: InstanceOfName IEC_TIMER
"IEC_TIMER"
BEGIN
END_DATA_BLOCK

DATA_BLOCK "IEC_Timer_CrossroadCycle_DB_1"   // DB10
{ S7_Optimized_Access := 'TRUE' }
AUTHOR : Simatic
FAMILY : IEC
NAME : IEC_TMR
VERSION : 1.0
// stored: InstanceOfName IEC_TIMER
"IEC_TIMER"
BEGIN
END_DATA_BLOCK

// folder: (top level)

ORGANIZATION_BLOCK "Main"   // OB1, LAD, ProgramCycle
TITLE = "Main Program Sweep (Cycle)"
{ S7_Optimized_Access := 'TRUE' }
VERSION : 0.1
   VAR_INPUT
      Initial_Call : Bool;   // Initial call of this OB
      Remanence : Bool;   // =True, if remanent data are available
   END_VAR
BEGIN

REGION Network 1: CarLight
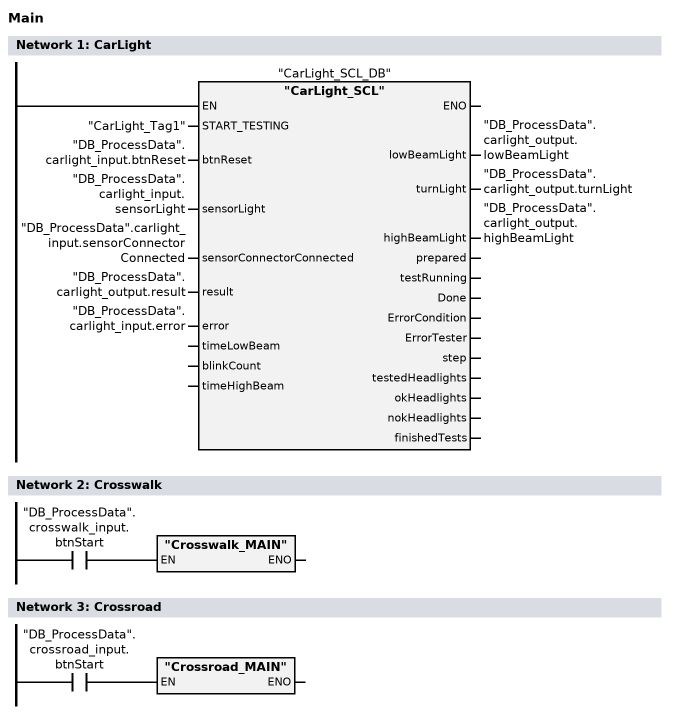
   RUNG wire#powerrail
      "CarLight_SCL_DB"(START_TESTING := "CarLight_Tag1", btnReset := "DB_ProcessData".carlight_input.btnReset, sensorLight := "DB_ProcessData".carlight_input.sensorLight, sensorConnectorConnected := "DB_ProcessData".carlight_input.sensorConnectorConnected, result := "DB_ProcessData".carlight_output.result, error := "DB_ProcessData".carlight_input.error, timeLowBeam :=, blinkCount :=, timeHighBeam :=, lowBeamLight => "DB_ProcessData".carlight_output.lowBeamLight, turnLight => "DB_ProcessData".carlight_output.turnLight, highBeamLight => "DB_ProcessData".carlight_output.highBeamLight, prepared =>, testRunning =>, Done =>, ErrorCondition =>, ErrorTester =>, "step" =>, testedHeadlights =>, okHeadlights =>, nokHeadlights =>, finishedTests =>)
   END_RUNG
   // the same network as SCL:
   "CarLight_SCL_DB"(START_TESTING := "CarLight_Tag1",   // "CarLight_SCL"
                     btnReset := "DB_ProcessData".carlight_input.btnReset,
                     sensorLight := "DB_ProcessData".carlight_input.sensorLight,
                     sensorConnectorConnected := "DB_ProcessData".carlight_input.sensorConnectorConnected,
                     result := "DB_ProcessData".carlight_output.result,
                     error := "DB_ProcessData".carlight_input.error,
                     lowBeamLight => "DB_ProcessData".carlight_output.lowBeamLight,
                     turnLight => "DB_ProcessData".carlight_output.turnLight,
                     highBeamLight => "DB_ProcessData".carlight_output.highBeamLight);
END_REGION

REGION Network 2: Crosswalk
   RUNG wire#powerrail
      Contact( "DB_ProcessData".crosswalk_input.btnStart )
      "Crosswalk_MAIN"()
   END_RUNG
   // the same network as SCL:
   IF "DB_ProcessData".crosswalk_input.btnStart THEN "Crosswalk_MAIN"(); END_IF;
END_REGION

REGION Network 3: Crossroad
   RUNG wire#powerrail
      Contact( "DB_ProcessData".crossroad_input.btnStart )
      "Crossroad_MAIN"()
   END_RUNG
   // the same network as SCL:
   IF "DB_ProcessData".crossroad_input.btnStart THEN "Crossroad_MAIN"(); END_IF;
END_REGION
END_ORGANIZATION_BLOCK

ORGANIZATION_BLOCK "CyclicInterrupt"   // OB30, LAD, CyclicInterrupt
{ S7_Optimized_Access := 'TRUE' }
VERSION : 0.1
   VAR_INPUT
      Initial_Call : Bool;   // Initial call of this OB
      Event_Count : Int;   // Events discarded
   END_VAR
BEGIN

REGION Network 1: Regulator
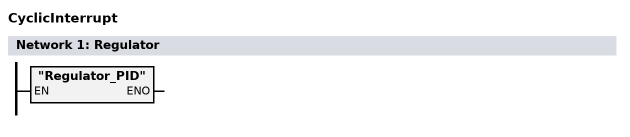
   RUNG wire#powerrail
      "Regulator_PID"()
   END_RUNG
   // the same network as SCL:
   "Regulator_PID"();
END_REGION
END_ORGANIZATION_BLOCK

ORGANIZATION_BLOCK "Startup"   // OB100, LAD, Startup
TITLE = "Complete Restart"
{ S7_Optimized_Access := 'TRUE' }
VERSION : 0.1
   VAR_INPUT
      LostRetentive : Bool;   // True if retentive data are lost
      LostRTC : Bool;   // True if date and time are lost
   END_VAR
BEGIN

REGION Network 1 (SCL)
   // Communication 


   // Crossroad
   "Crossorad_HoursDayStart" := 0;
   "Crossroad_HoursDayEnd" := 2400;
   "Crossroad_DayStarts" := 500;
   "Crossroad_DayEnds" := 2200;
   "Crossroad_S1" := 1;
   "Crossroad_S2" := 2;
   "Crossroad_S3" := 3;
   "Crossroad_S4" := 4;
   "Crossroad_S5" := 5;
   "Crossroad_S6" := 6;
   "Crossroad_S7" := 7;
   "Crossroad_S8" := 8;
   "Crossroad_S9" := 9;


   // Crosswalk


   // Regulaotr


   // CarLight
END_REGION
END_ORGANIZATION_BLOCK

// folder: CarLight

FUNCTION_BLOCK "CarLight_SCL"   // FB1, SCL
{ S7_Optimized_Access := 'TRUE' }
VERSION : 0.1
   VAR_INPUT
      START_TESTING : Bool;
      btnReset : Bool;
      sensorLight : Bool;
      sensorConnectorConnected : Bool;
      result : Bool;
      error : Bool;
      timeLowBeam : Time;
      blinkCount : Int;
      timeHighBeam : Time;
   END_VAR
   VAR_OUTPUT
      lowBeamLight : Bool;
      turnLight : Bool;
      highBeamLight : Bool;
      prepared : Bool;
      testRunning : Bool;
      Done : Bool;
      ErrorCondition : Bool;
      ErrorTester : Bool;
      "step" : Int;
      testedHeadlights : DInt;
      okHeadlights : DInt;
      nokHeadlights : DInt;
      finishedTests : DInt;
   END_VAR
   VAR
      state : Int;
      ready : Bool;
      start_old : Bool;
      start_rise : Bool;
      conditionsErrorLatched : Bool;
      testerErrorLatched : Bool;
      blinkTarget : Int;
      blinkIndex : Int;
      resultStored : Bool;
      testerResponseSeenTrue : Bool;
      tonLowBeam : TON_TIME;
      tonBlinkOn : TON_TIME;
      tonBlinkOff : TON_TIME;
      tonHighBeam : TON_TIME;
      tonAll : TON_TIME;
      tonTesterResponse : TON_TIME;
   END_VAR
BEGIN
   // ---------------------------------------------------------------------
   // Helper signals
   // ---------------------------------------------------------------------
   #ready := #sensorLight AND #sensorConnectorConnected;

   IF #blinkCount < 1 THEN
       #blinkTarget := 1;
   ELSE
       #blinkTarget := #blinkCount;
   END_IF;

   #start_rise := #START_TESTING AND NOT #start_old;
   #start_old := #START_TESTING;


   // ---------------------------------------------------------------------
   // RESET process (counters are NOT cleared)
   // ---------------------------------------------------------------------
   IF #btnReset THEN
       #state := 0;
       #conditionsErrorLatched := FALSE;
       #testerErrorLatched := FALSE;
       #blinkIndex := 0;
       #resultStored := FALSE;
       #testerResponseSeenTrue := FALSE;
   END_IF;


   // ---------------------------------------------------------------------
   // Loss of required conditions during test
   // ---------------------------------------------------------------------
   IF ((#state >= 20) AND (#state <= 55)) AND (NOT #ready) THEN
       #state := 0;
       #conditionsErrorLatched := TRUE;
       #blinkIndex := 0;
       #resultStored := FALSE;
       #testerResponseSeenTrue := FALSE;
   END_IF;


   // ---------------------------------------------------------------------
   // Tester error – immediate NOK termination
   // ---------------------------------------------------------------------
   IF ((#state >= 20) AND (#state <= 55)) AND #error THEN

       #testerErrorLatched := TRUE;

       IF NOT #resultStored THEN
           #testedHeadlights := #testedHeadlights + 1;
           #nokHeadlights := #nokHeadlights + 1;
           #resultStored := TRUE;
       END_IF;

       #blinkIndex := 0;
       #testerResponseSeenTrue := FALSE;

       #state := 70;

   END_IF;


   // ---------------------------------------------------------------------
   // State machine
   // ---------------------------------------------------------------------
   CASE #state OF


           // ==============================================================
           // 0 - IDLE
           // ==============================================================
       0:

           #lowBeamLight := FALSE;
           #turnLight := FALSE;
           #highBeamLight := FALSE;

           #tonLowBeam(IN := FALSE,
                     PT := #timeLowBeam);
           #tonBlinkOn(IN := FALSE,
                       PT := T#1s);
           #tonBlinkOff(IN := FALSE,
                        PT := T#1s);
           #tonHighBeam(IN := FALSE,
                     PT := #timeHighBeam);
           #tonAll(IN := FALSE,
                   PT := T#5s);
           #tonTesterResponse(IN := FALSE,
                              PT := T#1s);

           IF #start_rise THEN

               IF #ready AND (NOT #error) THEN

                   #conditionsErrorLatched := FALSE;
                   #testerErrorLatched := FALSE;
                   #blinkIndex := 0;
                   #resultStored := FALSE;
                   #testerResponseSeenTrue := FALSE;

                   #state := 20;

               ELSE

                   IF NOT #ready THEN
                       #conditionsErrorLatched := TRUE;
                   END_IF;

                   IF #error THEN
                       #testerErrorLatched := TRUE;
                   END_IF;

               END_IF;

           END_IF;


           // ==============================================================
           // 20 - LOW BEAM
           // ==============================================================
       20:

           #lowBeamLight := TRUE;
           #turnLight := FALSE;
           #highBeamLight := FALSE;

           #tonLowBeam(IN := TRUE,
                     PT := #timeLowBeam);
           #tonBlinkOn(IN := FALSE,
                       PT := T#1s);
           #tonBlinkOff(IN := FALSE,
                        PT := T#1s);
           #tonHighBeam(IN := FALSE,
                     PT := #timeHighBeam);
           #tonAll(IN := FALSE,
                   PT := T#5s);
           #tonTesterResponse(IN := FALSE,
                              PT := T#1s);

           IF #tonLowBeam.Q THEN
               #blinkIndex := 0;
               #state := 30;
           END_IF;


           // ==============================================================
           // 30 - TURN SIGNAL ON
           // ==============================================================
       30:

           #lowBeamLight := FALSE;
           #turnLight := TRUE;
           #highBeamLight := FALSE;

           #tonLowBeam(IN := FALSE,
                     PT := #timeLowBeam);
           #tonBlinkOn(IN := TRUE,
                       PT := T#1s);
           #tonBlinkOff(IN := FALSE,
                        PT := T#1s);
           #tonHighBeam(IN := FALSE,
                     PT := #timeHighBeam);
           #tonAll(IN := FALSE,
                   PT := T#5s);
           #tonTesterResponse(IN := FALSE,
                              PT := T#1s);

           IF #tonBlinkOn.Q THEN
               #state := 31;
           END_IF;


           // ==============================================================
           // 31 - TURN SIGNAL OFF
           // ==============================================================
       31:

           #lowBeamLight := FALSE;
           #turnLight := FALSE;
           #highBeamLight := FALSE;

           #tonLowBeam(IN := FALSE,
                     PT := #timeLowBeam);
           #tonBlinkOn(IN := FALSE,
                       PT := T#1s);
           #tonBlinkOff(IN := TRUE,
                        PT := T#1s);
           #tonHighBeam(IN := FALSE,
                     PT := #timeHighBeam);
           #tonAll(IN := FALSE,
                   PT := T#5s);
           #tonTesterResponse(IN := FALSE,
                              PT := T#1s);

           IF #tonBlinkOff.Q THEN

               #blinkIndex := #blinkIndex + 1;

               IF #blinkIndex < #blinkTarget THEN
                   #state := 30;
               ELSE
                   #state := 40;
               END_IF;

           END_IF;


           // ==============================================================
           // 40 - HIGH BEAM
           // ==============================================================
       40:

           #lowBeamLight := FALSE;
           #turnLight := FALSE;
           #highBeamLight := TRUE;

           #tonLowBeam(IN := FALSE,
                     PT := #timeLowBeam);
           #tonBlinkOn(IN := FALSE,
                       PT := T#1s);
           #tonBlinkOff(IN := FALSE,
                        PT := T#1s);
           #tonHighBeam(IN := TRUE,
                     PT := #timeHighBeam);
           #tonAll(IN := FALSE,
                   PT := T#5s);
           #tonTesterResponse(IN := FALSE,
                              PT := T#1s);

           IF #tonHighBeam.Q THEN
               #state := 50;
           END_IF;


           // ==============================================================
           // 50 - ALL LIGHTS (5 seconds)
           // ==============================================================
       50:

           #lowBeamLight := TRUE;
           #turnLight := TRUE;
           #highBeamLight := TRUE;

           #tonLowBeam(IN := FALSE,
                     PT := #timeLowBeam);
           #tonBlinkOn(IN := FALSE,
                       PT := T#1s);
           #tonBlinkOff(IN := FALSE,
                        PT := T#1s);
           #tonHighBeam(IN := FALSE,
                     PT := #timeHighBeam);
           #tonAll(IN := TRUE,
                   PT := T#5s);
           #tonTesterResponse(IN := FALSE,
                              PT := T#1s);

           IF #tonAll.Q THEN
               #testerResponseSeenTrue := FALSE;
               #state := 55;
           END_IF;


           // ==============================================================
           // 55 - WAIT 1 s FOR RESULT
           // ==============================================================
       55:

           #lowBeamLight := FALSE;
           #turnLight := FALSE;
           #highBeamLight := FALSE;

           #tonLowBeam(IN := FALSE,
                     PT := #timeLowBeam);
           #tonBlinkOn(IN := FALSE,
                       PT := T#1s);
           #tonBlinkOff(IN := FALSE,
                        PT := T#1s);
           #tonHighBeam(IN := FALSE,
                     PT := #timeHighBeam);
           #tonAll(IN := FALSE,
                   PT := T#5s);
           #tonTesterResponse(IN := TRUE,
                              PT := T#1s);

           IF #result THEN
               #testerResponseSeenTrue := TRUE;
           END_IF;

           IF #tonTesterResponse.Q THEN

               IF NOT #resultStored THEN

                   #testedHeadlights := #testedHeadlights + 1;

                   IF #testerResponseSeenTrue THEN
                       #okHeadlights := #okHeadlights + 1;
                   ELSE
                       #nokHeadlights := #nokHeadlights + 1;
                   END_IF;

                   #resultStored := TRUE;

               END_IF;

               #finishedTests := #finishedTests + 1;

               #state := 60;

           END_IF;


           // ==============================================================
           // 60 - FINISHED
           // ==============================================================
       60:

           #lowBeamLight := FALSE;
           #turnLight := FALSE;
           #highBeamLight := FALSE;

           IF #start_rise THEN

               IF #ready AND (NOT #error) THEN

                   #conditionsErrorLatched := FALSE;
                   #testerErrorLatched := FALSE;
                   #blinkIndex := 0;
                   #resultStored := FALSE;
                   #testerResponseSeenTrue := FALSE;

                   #state := 20;

               END_IF;

           END_IF;


           // ==============================================================
           // 70 - TESTER ERROR
           // ==============================================================
       70:

           #lowBeamLight := FALSE;
           #turnLight := FALSE;
           #highBeamLight := FALSE;

           IF #start_rise THEN

               IF #ready AND (NOT #error) THEN

                   #conditionsErrorLatched := FALSE;
                   #testerErrorLatched := FALSE;
                   #blinkIndex := 0;
                   #resultStored := FALSE;
                   #testerResponseSeenTrue := FALSE;

                   #state := 20;

               END_IF;

           END_IF;

       ELSE

           #state := 0;

   END_CASE;


   // ---------------------------------------------------------------------
   // State outputs
   // ---------------------------------------------------------------------
   #testRunning := (#state >= 20) AND (#state <= 55);

   #prepared := #ready AND (NOT #error) AND
   ((#state = 0) OR (#state = 60) OR (#state = 70));

   #Done := (#state = 60);

   #ErrorCondition := #conditionsErrorLatched;
   #ErrorTester := #testerErrorLatched;

   #step := #state;
END_FUNCTION_BLOCK

// folder: Crossroad

FUNCTION "Crossroad_MAIN" : Void   // FC4, LAD
{ S7_Optimized_Access := 'TRUE' }
VERSION : 0.1
   VAR_TEMP   // added for the SCL form of the ladder/FBD networks
      _w1 : Bool;
      _w2 : Bool;
      _w3 : Bool;
      _w4 : Bool;
   END_VAR
BEGIN

